KUKA KRL program: MyProgram_146().src

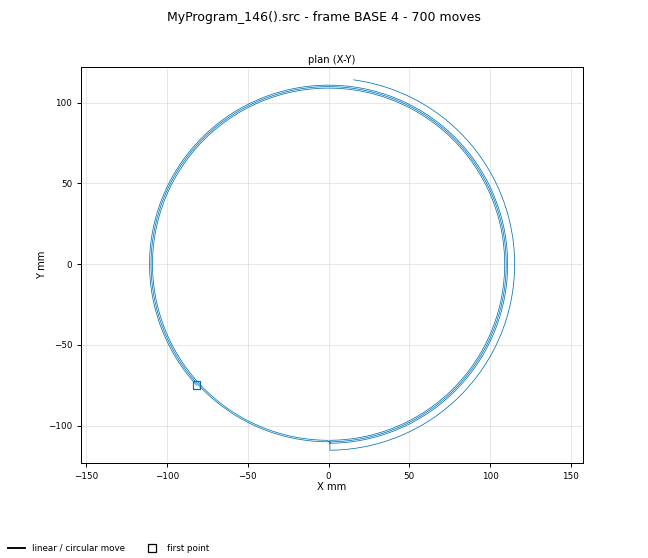
[picture p0: tool path of MyProgram_146().src in frame BASE 4, 700 of 700 moves have a stored position in this frame; points joined in program order, loops and branches not executed]
&ACCESS RVP
&REL 1
&PARAM TEMPLATE = C:\KRC\Roboter\Template\vorgabe
&PARAM EDITMASK = *
DEF MyProgram_146()
; ---- Setting reference (Base) ----
$BASE = BASE_DATA[4]

; --------------------------
; ---- Setting tool (TCP) ----
$TOOL = TOOL_DATA[3]
; --------------------------

$VEL.CP = VEL_APROX_PRINT
Startdeposition()
$VEL.CP = VEL_PRINT
LIN {X -81.7573,Y -74.8316,Z 115,A -141.7153,B 24.9501,C -1.6313,E1 24.8814,E2 227.6019} C_DIS
LIN {X -84.7818,Y -71.3896,Z 115,A -144.2948,B 24.9503,C -1.6285,E1 24.8767,E2 230.1997} C_DIS
LIN {X -86.9243,Y -68.7617,Z 115,A -146.5277,B 24.9512,C -1.6142,E1 24.8727,E2 232.4772} C_DIS
LIN {X -89.3897,Y -65.5248,Z 115,A -148.18,B 24.9498,C -1.6368,E1 24.87,E2 234.0837} C_DIS
LIN {X -91.5986,Y -62.4003,Z 115,A -150.3386,B 24.9499,C -1.6348,E1 24.8666,E2 236.2576} C_DIS
LIN {X -94.0442,Y -58.649,Z 115,A -152.3948,B 24.9489,C -1.6509,E1 24.8635,E2 238.286} C_DIS
LIN {X -96.0088,Y -55.3746,Z 115,A -154.4318,B 24.9488,C -1.6537,E1 24.8607,E2 240.3268} C_DIS
LIN {X -98.582,Y -50.6523,Z 115,A -157.2694,B 24.9484,C -1.6592,E1 24.8569,E2 243.1663} C_DIS
LIN {X -100.3639,Y -47.023,Z 115,A -159.3857,B 24.9481,C -1.6641,E1 24.8544,E2 245.2824} C_DIS
LIN {X -102.0957,Y -43.1333,Z 115,A -161.4118,B 24.9473,C -1.6772,E1 24.8521,E2 247.2885} C_DIS
LIN {X -103.2527,Y -40.2858,Z 115,A -163.0662,B 24.9472,C -1.6793,E1 24.8504,E2 248.9471} C_DIS
LIN {X -104.2802,Y -37.548,Z 115,A -164.6637,B 24.9471,C -1.6805,E1 24.8489,E2 250.5507} C_DIS
LIN {X -105.4561,Y -34.1032,Z 115,A -166.5332,B 24.9467,C -1.6867,E1 24.8472,E2 252.4164} C_DIS
LIN {X -107.1592,Y -28.3073,Z 115,A -169.7153,B 24.9462,C -1.6939,E1 24.8448,E2 255.5995} C_DIS
LIN {X -108.4327,Y -22.9525,Z 115,A -172.6096,B 24.9458,C -1.7009,E1 24.843,E2 258.4941} C_DIS
LIN {X -108.951,Y -20.3482,Z 115,A -173.8603,B 24.9452,C -1.7099,E1 24.8423,E2 259.7309} C_DIS
LIN {X -109.5336,Y -16.923,Z 115,A -175.6733,B 24.9449,C -1.7149,E1 24.8415,E2 261.5426} C_DIS
LIN {X -110.023,Y -13.3864,Z 115,A -177.655,B 24.9449,C -1.7156,E1 24.8408,E2 263.5345} C_DIS
LIN {X -110.406,Y -9.7333,Z 115,A -179.5845,B 24.9445,C -1.7206,E1 24.8403,E2 265.4638} C_DIS
LIN {X -110.6566,Y -6.2558,Z 115,A 178.7094,B 24.9439,C -1.73,E1 24.84,E2 267.1575} C_DIS
LIN {X -110.8019,Y -2.7097,Z 115,A 176.7644,B 24.9438,C -1.7318,E1 24.8398,E2 269.1101} C_DIS
LIN {X -110.8276,Y 1.2801,Z 115,A 174.684,B 24.9434,C -1.7378,E1 24.8398,E2 271.1887} C_DIS
LIN {X -110.7364,Y 4.6333,Z 115,A 173.0527,B 24.9428,C -1.7473,E1 24.84,E2 272.807} C_DIS
LIN {X -110.534,Y 8.1638,Z 115,A 171.0925,B 24.9428,C -1.7483,E1 24.8403,E2 274.7769} C_DIS
LIN {X -110.2005,Y 11.8298,Z 115,A 169.1643,B 24.9424,C -1.7535,E1 24.8409,E2 276.7041} C_DIS
LIN {X -109.6262,Y 16.3247,Z 115,A 166.4672,B 24.9428,C -1.7477,E1 24.8419,E2 279.431} C_DIS
LIN {X -109.0594,Y 19.7502,Z 115,A 164.6359,B 24.9425,C -1.7522,E1 24.8428,E2 281.2625} C_DIS
LIN {X -108.342,Y 23.3687,Z 115,A 163.4659,B 24.9402,C -1.7861,E1 24.8435,E2 282.3586} C_DIS
LIN {X -106.823,Y 29.5519,Z 115,A 159.9331,B 24.9402,C -1.7874,E1 24.8459,E2 285.909} C_DIS
LIN {X -105.5105,Y 33.9351,Z 115,A 157.4846,B 24.9398,C -1.7917,E1 24.8479,E2 288.3612} C_DIS
LIN {X -104.4742,Y 37.0035,Z 115,A 155.7145,B 24.9398,C -1.7934,E1 24.8495,E2 290.1375} C_DIS
LIN {X -103.1875,Y 40.4518,Z 115,A 154.094,B 24.9386,C -1.81,E1 24.8511,E2 291.7276} C_DIS
LIN {X -100.9318,Y 45.7915,Z 115,A 150.7623,B 24.9388,C -1.8064,E1 24.8548,E2 295.0862} C_DIS
LIN {X -99.2356,Y 49.3592,Z 115,A 148.8447,B 24.9381,C -1.8172,E1 24.8571,E2 296.9882} C_DIS
LIN {X -97.7685,Y 52.2085,Z 115,A 147.0374,B 24.9381,C -1.8164,E1 24.8595,E2 298.8072} C_DIS
LIN {X -96.07,Y 55.2682,Z 115,A 145.1429,B 24.9381,C -1.8185,E1 24.8621,E2 300.7066} C_DIS
LIN {X -92.0549,Y 61.7265,Z 115,A 141.3379,B 24.9369,C -1.8344,E1 24.8678,E2 304.4929} C_DIS
LIN {X -90.3878,Y 64.1416,Z 115,A 139.117,B 24.9385,C -1.812,E1 24.8715,E2 306.7782} C_DIS
LIN {X -87.5356,Y 67.9832,Z 115,A 137.571,B 24.9356,C -1.8539,E1 24.8739,E2 308.2317} C_DIS
LIN {X -83.6667,Y 72.6909,Z 115,A 134.1861,B 24.9356,C -1.8531,E1 24.88,E2 311.6341} C_DIS
LIN {X -79.1475,Y 77.5878,Z 115,A 129.9553,B 24.9371,C -1.8317,E1 24.8883,E2 315.9343} C_DIS
LIN {X -75.6083,Y 81.0407,Z 115,A 128.058,B 24.9349,C -1.8629,E1 24.892,E2 317.765} C_DIS
LIN {X -70.4692,Y 85.5472,Z 115,A 123.8886,B 24.9361,C -1.8465,E1 24.901,E2 321.9897} C_DIS
LIN {X -66.7924,Y 88.4469,Z 115,A 122.3719,B 24.9333,C -1.8865,E1 24.9041,E2 323.4166} C_DIS
LIN {X -62.2506,Y 91.7,Z 115,A 119.1568,B 24.9338,C -1.8796,E1 24.9115,E2 326.6592} C_DIS
LIN {X -58.8492,Y 93.9192,Z 115,A 117.1695,B 24.9332,C -1.888,E1 24.9162,E2 328.6329} C_DIS
LIN {X -56.138,Y 95.5648,Z 115,A 115.439,B 24.9332,C -1.8874,E1 24.9203,E2 330.37} C_DIS
LIN {X -53.5767,Y 97.0249,Z 115,A 113.3768,B 24.9345,C -1.8691,E1 24.9255,E2 332.4818} C_DIS
LIN {X -49.7768,Y 99.0286,Z 115,A 111.6694,B 24.9328,C -1.8928,E1 24.9296,E2 334.1375} C_DIS
LIN {X -46.6238,Y 100.5498,Z 115,A 110.0445,B 24.9321,C -1.9029,E1 24.9337,E2 335.7423} C_DIS
LIN {X -40.112,Y 103.321,Z 115,A 106.2146,B 24.9322,C -1.9013,E1 24.9436,E2 339.5847} C_DIS
LIN {X -35.6021,Y 104.9597,Z 115,A 103.1863,B 24.9335,C -1.8828,E1 24.9517,E2 342.6629} C_DIS
LIN {X -31.5857,Y 106.2373,Z 115,A 101.555,B 24.9318,C -1.907,E1 24.9559,E2 344.2396} C_DIS
LIN {X -26.5277,Y 107.6121,Z 115,A 98.9611,B 24.9313,C -1.9143,E1 24.9629,E2 346.82} C_DIS
LIN {X -23.7708,Y 108.2542,Z 115,A 97.4433,B 24.9313,C -1.9135,E1 24.967,E2 348.3417} C_DIS
LIN {X -20.5939,Y 108.9038,Z 115,A 95.6798,B 24.9315,C -1.9113,E1 24.9718,E2 350.1123} C_DIS
LIN {X -16.923,Y 109.5336,Z 115,A 93.8834,B 24.931,C -1.9179,E1 24.9768,E2 351.8948} C_DIS
LIN {X -13.8535,Y 109.9647,Z 115,A 92.371,B 24.9307,C -1.9226,E1 24.9809,E2 353.3972} C_DIS
LIN {X -10.0487,Y 110.3769,Z 115,A 90.2727,B 24.931,C -1.9187,E1 24.9868,E2 355.5058} C_DIS
LIN {X -6.4735,Y 110.6446,Z 115,A 88.3325,B 24.9312,C -1.916,E1 24.9922,E2 357.4533} C_DIS
LIN {X -3.889,Y 110.7661,Z 115,A 86.8091,B 24.9317,C -1.9088,E1 24.9965,E2 358.9939} C_DIS
LIN {X 0.2371,Y 110.8339,Z 115,A 84.7338,B 24.9315,C -1.9116,E1 25.0023,E2 361.0626} C_DIS
LIN {X 4.4661,Y 110.7436,Z 115,A 82.7039,B 24.931,C -1.9183,E1 25.0079,E2 363.0763} C_DIS
LIN {X 7.7943,Y 110.5593,Z 115,A 80.9252,B 24.9312,C -1.916,E1 25.0129,E2 364.8597} C_DIS
LIN {X 11.1548,Y 110.2712,Z 115,A 79.1362,B 24.9313,C -1.9139,E1 25.0178,E2 366.6525} C_DIS
LIN {X 15.2675,Y 109.7771,Z 115,A 77.1238,B 24.931,C -1.9188,E1 25.0234,E2 368.6517} C_DIS
LIN {X 18.2241,Y 109.3247,Z 115,A 75.5914,B 24.931,C -1.9188,E1 25.0276,E2 370.1824} C_DIS
LIN {X 21.6751,Y 108.6949,Z 115,A 73.7246,B 24.9312,C -1.9159,E1 25.0327,E2 372.0541} C_DIS
LIN {X 24.7884,Y 108.0258,Z 115,A 72.0718,B 24.9312,C -1.9148,E1 25.0372,E2 373.7073} C_DIS
LIN {X 28.6398,Y 107.0694,Z 115,A 69.2783,B 24.9336,C -1.8827,E1 25.045,E2 376.5725} C_DIS
LIN {X 33.4912,Y 105.6541,Z 115,A 67.5311,B 24.9311,C -1.9167,E1 25.0494,E2 378.236} C_DIS
LIN {X 37.5394,Y 104.2834,Z 115,A 65.2305,B 24.9315,C -1.9109,E1 25.0555,E2 380.5457} C_DIS
LIN {X 40.4462,Y 103.1897,Z 115,A 63.6357,B 24.9316,C -1.9098,E1 25.0597,E2 382.1396} C_DIS
LIN {X 43.8995,Y 101.7695,Z 115,A 61.6688,B 24.9319,C -1.9062,E1 25.0647,E2 384.1106} C_DIS
LIN {X 46.9047,Y 100.419,Z 115,A 59.6955,B 24.9328,C -1.8927,E1 25.0698,E2 386.1106} C_DIS
LIN {X 51.8783,Y 97.9424,Z 115,A 56.88,B 24.9329,C -1.8914,E1 25.0768,E2 388.9215} C_DIS
LIN {X 56.568,Y 95.3106,Z 115,A 54.359,B 24.9324,C -1.8984,E1 25.0828,E2 391.4183} C_DIS
LIN {X 59.6032,Y 93.4429,Z 115,A 52.5572,B 24.9325,C -1.8973,E1 25.0871,E2 393.2171} C_DIS
LIN {X 62.4108,Y 91.5915,Z 115,A 50.819,B 24.9327,C -1.8944,E1 25.0911,E2 394.9561} C_DIS
LIN {X 65.368,Y 89.5045,Z 115,A 49.1942,B 24.9322,C -1.9018,E1 25.0948,E2 396.5578} C_DIS
LIN {X 67.3354,Y 88.0347,Z 115,A 47.6455,B 24.9332,C -1.8875,E1 25.0983,E2 398.1348} C_DIS
LIN {X 69.5282,Y 86.313,Z 115,A 46.1298,B 24.9336,C -1.8816,E1 25.1016,E2 399.6588} C_DIS
LIN {X 72.7487,Y 83.6163,Z 115,A 44.0933,B 24.9336,C -1.8832,E1 25.1059,E2 401.6836} C_DIS
LIN {X 76.092,Y 80.5858,Z 115,A 41.7552,B 24.9339,C -1.8782,E1 25.1107,E2 404.024} C_DIS
LIN {X 78.6426,Y 78.0989,Z 115,A 40.1113,B 24.9335,C -1.8829,E1 25.114,E2 405.65} C_DIS
LIN {X 82.0766,Y 74.4837,Z 115,A 37.2578,B 24.9348,C -1.865,E1 25.1195,E2 408.5332} C_DIS
LIN {X 84.4274,Y 71.8056,Z 115,A 35.5078,B 24.9348,C -1.8648,E1 25.1226,E2 410.2757} C_DIS
LIN {X 86.8535,Y 68.8514,Z 115,A 33.7446,B 24.9345,C -1.8694,E1 25.1257,E2 412.0199} C_DIS
LIN {X 89.0528,Y 65.9849,Z 115,A 31.6509,B 24.9355,C -1.8548,E1 25.1293,E2 414.138} C_DIS
LIN {X 90.925,Y 63.3772,Z 115,A 30.0629,B 24.9355,C -1.8538,E1 25.1318,E2 415.7207} C_DIS
LIN {X 92.9023,Y 60.4452,Z 115,A 28.1746,B 24.9361,C -1.8464,E1 25.1348,E2 417.6171} C_DIS
LIN {X 95.8988,Y 55.566,Z 115,A 24.8642,B 24.9377,C -1.8231,E1 25.1396,E2 420.9656} C_DIS
LIN {X 97.6104,Y 52.5013,Z 115,A 23.4849,B 24.9367,C -1.8373,E1 25.1414,E2 422.3042} C_DIS
LIN {X 99.1431,Y 49.5458,Z 115,A 21.7653,B 24.9371,C -1.8325,E1 25.1435,E2 424.0259} C_DIS
LIN {X 100.5688,Y 46.5828,Z 115,A 20.112,B 24.9372,C -1.8297,E1 25.1455,E2 425.6768} C_DIS
LIN {X 102.0077,Y 43.3421,Z 115,A 18.1675,B 24.9379,C -1.8195,E1 25.1477,E2 427.6349} C_DIS
LIN {X 104.8831,Y 35.8293,Z 115,A 14.3206,B 24.9379,C -1.821,E1 25.1514,E2 431.4568} C_DIS
LIN {X 106.5349,Y 30.5691,Z 115,A 11.3263,B 24.9389,C -1.8058,E1 25.1539,E2 434.4698} C_DIS
LIN {X 107.3131,Y 27.7113,Z 115,A 9.7848,B 24.9392,C -1.8007,E1 25.155,E2 436.0146} C_DIS
LIN {X 108.1774,Y 24.1233,Z 115,A 7.8397,B 24.9397,C -1.793,E1 25.1562,E2 437.9664} C_DIS
LIN {X 108.884,Y 20.697,Z 115,A 5.995,B 24.9402,C -1.7857,E1 25.1572,E2 439.8175} C_DIS
LIN {X 109.5415,Y 16.8721,Z 115,A 4.1105,B 24.9402,C -1.7848,E1 25.1581,E2 441.6932} C_DIS
LIN {X 110.0434,Y 13.2119,Z 115,A 2.0838,B 24.9411,C -1.7735,E1 25.1588,E2 443.7346} C_DIS
LIN {X 110.4516,Y 9.1978,Z 115,A 0.0951,B 24.9412,C -1.7711,E1 25.1593,E2 445.7171} C_DIS
LIN {X 110.6876,Y 5.6966,Z 115,A -1.8682,B 24.942,C -1.7586,E1 25.1597,E2 447.6983} C_DIS
LIN {X 110.8179,Y 1.8536,Z 115,A -3.8981,B 24.9426,C -1.7502,E1 25.1597,E2 449.7357} C_DIS
LIN {X 110.7895,Y -3.1254,Z 115,A -6.2103,B 24.9424,C -1.7536,E1 25.1597,E2 452.0262} C_DIS
LIN {X 110.6672,Y -6.0644,Z 115,A -8.3066,B 24.9444,C -1.7229,E1 25.1594,E2 454.1824} C_DIS
LIN {X 110.3562,Y -10.2724,Z 115,A -9.8676,B 24.943,C -1.7435,E1 25.159,E2 455.6856} C_DIS
LIN {X 109.9421,Y -14.0283,Z 115,A -11.804,B 24.9434,C -1.7379,E1 25.1584,E2 457.6237} C_DIS
LIN {X 109.5152,Y -17.0426,Z 115,A -13.3694,B 24.9437,C -1.7332,E1 25.1577,E2 459.1911} C_DIS
LIN {X 108.8663,Y -20.7887,Z 115,A -15.2807,B 24.944,C -1.7293,E1 25.1568,E2 461.1005} C_DIS
LIN {X 108.2063,Y -23.9905,Z 115,A -17.0194,B 24.9445,C -1.7216,E1 25.1558,E2 462.8471} C_DIS
LIN {X 107.4311,Y -27.2525,Z 115,A -18.7555,B 24.9448,C -1.7159,E1 25.1546,E2 464.5865} C_DIS
LIN {X 106.7672,Y -29.7492,Z 115,A -20.4664,B 24.9462,C -1.6949,E1 25.1533,E2 466.3373} C_DIS
LIN {X 105.817,Y -32.9666,Z 115,A -21.8898,B 24.9456,C -1.7033,E1 25.1521,E2 467.7328} C_DIS
LIN {X 104.6176,Y -36.5948,Z 115,A -23.6513,B 24.9454,C -1.7067,E1 25.1506,E2 469.4764} C_DIS
LIN {X 103.7534,Y -38.9785,Z 115,A -25.1912,B 24.9463,C -1.6923,E1 25.1491,E2 471.0416} C_DIS
LIN {X 102.2201,Y -42.8382,Z 115,A -27.182,B 24.9463,C -1.6926,E1 25.147,E2 473.0206} C_DIS
LIN {X 100.7679,Y -46.1551,Z 115,A -28.9646,B 24.9464,C -1.6909,E1 25.1449,E2 474.7976} C_DIS
LIN {X 98.7191,Y -50.3841,Z 115,A -31.9765,B 24.9485,C -1.6576,E1 25.1411,E2 477.8719} C_DIS
LIN {X 96.8713,Y -53.8517,Z 115,A -33.4559,B 24.9474,C -1.6762,E1 25.1392,E2 479.2998} C_DIS
LIN {X 95.5696,Y -56.1298,Z 115,A -35.2243,B 24.9487,C -1.6538,E1 25.1367,E2 481.1118} C_DIS
LIN {X 93.7863,Y -59.0619,Z 115,A -36.7745,B 24.9484,C -1.6587,E1 25.1344,E2 482.6427} C_DIS
LIN {X 90.7878,Y -63.5747,Z 115,A -39.4423,B 24.9486,C -1.6567,E1 25.1302,E2 485.3019} C_DIS
LIN {X 88.6944,Y -66.463,Z 115,A -41.1973,B 24.9486,C -1.6556,E1 25.1273,E2 487.0511} C_DIS
LIN {X 86.5166,Y -69.2771,Z 115,A -43.1288,B 24.9492,C -1.6465,E1 25.1239,E2 488.995} C_DIS
LIN {X 84.2505,Y -72.0131,Z 115,A -44.9007,B 24.9493,C -1.6446,E1 25.1208,E2 490.7634} C_DIS
LIN {X 81.7575,Y -74.8315,Z 115,A -46.8119,B 24.9495,C -1.6411,E1 25.1172,E2 492.6742} C_DIS
LIN {X 79.0371,Y -77.6995,Z 115,A -48.8035,B 24.9497,C -1.6383,E1 25.1133,E2 494.6639} C_DIS
LIN {X 76.7863,Y -79.9244,Z 115,A -50.4986,B 24.9501,C -1.6317,E1 25.1099,E2 496.3675} C_DIS
LIN {X 74.0477,Y -82.468,Z 115,A -52.3792,B 24.9502,C -1.6294,E1 25.1061,E2 498.2458} C_DIS
LIN {X 71.2837,Y -84.8704,Z 115,A -54.3202,B 24.9506,C -1.623,E1 25.1019,E2 500.1946} C_DIS
LIN {X 68.6576,Y -87.0066,Z 115,A -55.9786,B 24.9506,C -1.6231,E1 25.0983,E2 501.8463} C_DIS
LIN {X 65.6879,Y -89.2702,Z 115,A -57.9458,B 24.951,C -1.6174,E1 25.0939,E2 503.82} C_DIS
LIN {X 62.8535,Y -91.2891,Z 115,A -59.5768,B 24.9508,C -1.6211,E1 25.0902,E2 505.4367} C_DIS
LIN {X 60.4943,Y -92.87,Z 115,A -62.3586,B 24.9543,C -1.5612,E1 25.0834,E2 508.3508} C_DIS
LIN {X 54.7496,Y -96.368,Z 115,A -65.2533,B 24.9532,C -1.5799,E1 25.0765,E2 511.1928} C_DIS
LIN {X 50.9504,Y -98.4297,Z 115,A -66.9022,B 24.952,C -1.6013,E1 25.0726,E2 512.7863} C_DIS
LIN {X 47.5157,Y -100.1327,Z 115,A -68.9366,B 24.9523,C -1.5958,E1 25.0674,E2 514.8283} C_DIS
LIN {X 44.9116,Y -101.3283,Z 115,A -70.6659,B 24.9531,C -1.5828,E1 25.063,E2 516.584} C_DIS
LIN {X 40.4823,Y -103.1756,Z 115,A -72.88,B 24.9526,C -1.5908,E1 25.0573,E2 518.7742} C_DIS
LIN {X 35.6279,Y -104.951,Z 115,A -75.4422,B 24.9526,C -1.592,E1 25.0506,E2 521.3284} C_DIS
LIN {X 32.2394,Y -106.0419,Z 115,A -77.3857,B 24.9529,C -1.5854,E1 25.0454,E2 523.2841} C_DIS
LIN {X 28.9748,Y -106.9789,Z 115,A -79.0339,B 24.9527,C -1.5881,E1 25.041,E2 524.9231} C_DIS
LIN {X 25.2858,Y -107.9109,Z 115,A -81.0187,B 24.9529,C -1.5854,E1 25.0356,E2 526.9115} C_DIS
LIN {X 22.1944,Y -108.5883,Z 115,A -82.4818,B 24.9526,C -1.5913,E1 25.0316,E2 528.3588} C_DIS
LIN {X 18.4966,Y -109.2791,Z 115,A -84.5679,B 24.953,C -1.5837,E1 25.0258,E2 530.4605} C_DIS
LIN {X 15.2443,Y -109.7804,Z 115,A -86.3172,B 24.9532,C -1.5804,E1 25.021,E2 532.2159} C_DIS
LIN {X 12.7171,Y -110.1014,Z 115,A -87.747,B 24.9535,C -1.5749,E1 25.017,E2 533.6579} C_DIS
LIN {X 6.9538,Y -110.6161,Z 115,A -90.5923,B 24.9533,C -1.5795,E1 25.0091,E2 536.4906} C_DIS
LIN {X 3.5153,Y -110.7775,Z 115,A -92.3395,B 24.9533,C -1.5803,E1 25.0042,E2 538.2356} C_DIS
LIN {X 0.7828,Y -110.8248,Z 115,A -93.8199,B 24.9533,C -1.5771,E1 25.0001,E2 539.7233} C_DIS
Enddeposition()
LIN {X 0.7828,Y -110.8248,Z 115,A -93.8199,B 24.9533,C -1.5771,E1 25.0001,E2 539.7233} C_DIS
Startdeposition()
$VEL.CP = VEL_PRINT
LIN {X 1.4576,Y -109.912,Z 115,A -92.785,B 24.9507,C -1.6218,E1 25.0033,E2 538.5826} C_DIS
LIN {X 4.6673,Y -109.8211,Z 115,A -91.0978,B 24.9507,C -1.623,E1 25.008,E2 536.893} C_DIS
LIN {X 7.5586,Y -109.6601,Z 115,A -89.4834,B 24.9503,C -1.6281,E1 25.0125,E2 535.2672} C_DIS
LIN {X 11.1892,Y -109.3495,Z 115,A -87.5115,B 24.9501,C -1.6322,E1 25.018,E2 533.2868} C_DIS
LIN {X 14.8057,Y -108.9205,Z 115,A -85.5197,B 24.9498,C -1.6373,E1 25.0236,E2 531.2843} C_DIS
LIN {X 18.9126,Y -108.2823,Z 115,A -83.6444,B 24.9504,C -1.6265,E1 25.0287,E2 529.4365} C_DIS
LIN {X 22.0138,Y -107.6933,Z 115,A -81.8972,B 24.9501,C -1.6323,E1 25.0335,E2 527.6777} C_DIS
LIN {X 25.453,Y -106.9345,Z 115,A -79.9474,B 24.9497,C -1.6389,E1 25.0388,E2 525.7149} C_DIS
LIN {X 29.0229,Y -106.0201,Z 115,A -78.0363,B 24.9496,C -1.6406,E1 25.044,E2 523.8029} C_DIS
LIN {X 31.771,Y -105.2299,Z 115,A -76.3612,B 24.949,C -1.6503,E1 25.0485,E2 522.1078} C_DIS
LIN {X 36.3044,Y -103.7519,Z 115,A -73.5988,B 24.948,C -1.6655,E1 25.0559,E2 519.3147} C_DIS
LIN {X 40.1137,Y -102.3394,Z 115,A -71.6969,B 24.9484,C -1.659,E1 25.0608,E2 517.4325} C_DIS
LIN {X 43.1125,Y -101.1137,Z 115,A -70.4315,B 24.9494,C -1.6431,E1 25.0639,E2 516.2078} C_DIS
LIN {X 45.8081,Y -99.9224,Z 115,A -68.7252,B 24.9488,C -1.6528,E1 25.0683,E2 514.4827} C_DIS
LIN {X 48.7959,Y -98.4957,Z 115,A -67.0984,B 24.9488,C -1.6514,E1 25.0724,E2 512.8636} C_DIS
LIN {X 51.1648,Y -97.2863,Z 115,A -65.5915,B 24.9484,C -1.659,E1 25.0761,E2 511.3429} C_DIS
LIN {X 54.8199,Y -95.2745,Z 115,A -63.5622,B 24.9486,C -1.6565,E1 25.0811,E2 509.3255} C_DIS
LIN {X 58.1891,Y -93.255,Z 115,A -61.7581,B 24.949,C -1.6497,E1 25.0853,E2 507.5431} C_DIS
LIN {X 62.6693,Y -90.3051,Z 115,A -58.7684,B 24.9481,C -1.6637,E1 25.0923,E2 504.5302} C_DIS
LIN {X 65.4015,Y -88.3483,Z 115,A -56.9115,B 24.9476,C -1.672,E1 25.0965,E2 502.6603} C_DIS
LIN {X 68.1462,Y -86.247,Z 115,A -55.2231,B 24.9476,C -1.671,E1 25.1002,E2 500.9807} C_DIS
LIN {X 71.0085,Y -83.9069,Z 115,A -53.25,B 24.9473,C -1.6773,E1 25.1045,E2 499.0001} C_DIS
LIN {X 73.7158,Y -81.5397,Z 115,A -51.3437,B 24.9469,C -1.6831,E1 25.1085,E2 497.0877} C_DIS
LIN {X 76.198,Y -79.2233,Z 115,A -49.6701,B 24.9469,C -1.6831,E1 25.1118,E2 495.421} C_DIS
LIN {X 78.6653,Y -76.7767,Z 115,A -47.7296,B 24.9463,C -1.6933,E1 25.1157,E2 493.4647} C_DIS
LIN {X 81.2752,Y -74.0066,Z 115,A -45.7835,B 24.9461,C -1.6967,E1 25.1194,E2 491.5192} C_DIS
LIN {X 83.5964,Y -71.3731,Z 115,A -44.0758,B 24.9461,C -1.696,E1 25.1225,E2 489.8208} C_DIS
LIN {X 85.812,Y -68.6964,Z 115,A -42.1422,B 24.9454,C -1.7063,E1 25.1259,E2 487.8719} C_DIS
LIN {X 88.352,Y -65.3964,Z 115,A -40.0792,B 24.9454,C -1.7074,E1 25.1294,E2 485.8161} C_DIS
LIN {X 90.1847,Y -62.8426,Z 115,A -37.7884,B 24.9432,C -1.7414,E1 25.1331,E2 483.4563} C_DIS
LIN {X 92.7748,Y -58.9537,Z 115,A -36.0541,B 24.9448,C -1.7167,E1 25.1357,E2 481.7891} C_DIS
LIN {X 94.7217,Y -55.77,Z 115,A -34.1518,B 24.9445,C -1.7204,E1 25.1384,E2 479.8878} C_DIS
LIN {X 96.4518,Y -52.7223,Z 115,A -32.2608,B 24.944,C -1.7287,E1 25.141,E2 477.9871} C_DIS
LIN {X 97.7068,Y -50.3585,Z 115,A -30.3408,B 24.9422,C -1.7566,E1 25.1435,E2 476.0115} C_DIS
LIN {X 99.537,Y -46.6359,Z 115,A -28.7858,B 24.9435,C -1.7356,E1 25.1453,E2 474.5142} C_DIS
LIN {X 100.9223,Y -43.558,Z 115,A -27.0904,B 24.9434,C -1.7381,E1 25.1472,E2 472.8222} C_DIS
LIN {X 102.2903,Y -40.2388,Z 115,A -25.4454,B 24.9437,C -1.7338,E1 25.1489,E2 471.1965} C_DIS
LIN {X 103.8515,Y -36.0204,Z 115,A -22.9448,B 24.9427,C -1.7481,E1 25.1513,E2 468.6762} C_DIS
LIN {X 105.806,Y -29.7921,Z 115,A -19.4702,B 24.9418,C -1.7621,E1 25.1542,E2 465.1884} C_DIS
LIN {X 106.6681,Y -26.5449,Z 115,A -17.653,B 24.9412,C -1.7706,E1 25.1554,E2 463.3615} C_DIS
LIN {X 107.4491,Y -23.1778,Z 115,A -15.8685,B 24.9409,C -1.7757,E1 25.1565,E2 461.5754} C_DIS
LIN {X 108.1717,Y -19.5282,Z 115,A -14.0375,B 24.9409,C -1.777,E1 25.1575,E2 459.7519} C_DIS
LIN {X 108.6569,Y -16.6183,Z 115,A -12.448,B 24.9403,C -1.7844,E1 25.1582,E2 458.1545} C_DIS
LIN {X 109.1437,Y -13.0455,Z 115,A -10.6244,B 24.9401,C -1.788,E1 25.1588,E2 456.3332} C_DIS
LIN {X 109.4667,Y -9.975,Z 115,A -9.2078,B 24.9403,C -1.7845,E1 25.1592,E2 454.9332} C_DIS
LIN {X 109.6979,Y -6.9997,Z 115,A -7.3761,B 24.9391,C -1.802,E1 25.1596,E2 453.071} C_DIS
LIN {X 109.859,Y -3.6799,Z 115,A -5.9668,B 24.9397,C -1.7931,E1 25.1597,E2 451.6912} C_DIS
LIN {X 109.9189,Y -0.535,Z 115,A -4.0353,B 24.9385,C -1.8116,E1 25.1597,E2 449.7276} C_DIS
LIN {X 109.8898,Y 2.662,Z 115,A -2.2548,B 24.9378,C -1.8221,E1 25.1597,E2 447.9327} C_DIS
LIN {X 109.693,Y 7.0722,Z 115,A -0.2487,B 24.9382,C -1.8162,E1 25.1594,E2 445.9525} C_DIS
LIN {X 109.43,Y 10.3734,Z 115,A 1.6087,B 24.9374,C -1.8277,E1 25.1589,E2 444.079} C_DIS
LIN {X 109.0112,Y 14.1072,Z 115,A 3.4891,B 24.9372,C -1.8305,E1 25.1583,E2 442.2033} C_DIS
LIN {X 108.4782,Y 17.7505,Z 115,A 5.2562,B 24.9372,C -1.8297,E1 25.1576,E2 440.4483} C_DIS
LIN {X 108.0255,Y 20.3262,Z 115,A 6.7767,B 24.9365,C -1.8411,E1 25.1568,E2 438.9099} C_DIS
LIN {X 107.3718,Y 23.532,Z 115,A 8.436,B 24.9362,C -1.8444,E1 25.1558,E2 437.2525} C_DIS
LIN {X 106.5272,Y 27.1013,Z 115,A 10.2668,B 24.9361,C -1.8467,E1 25.1546,E2 435.4269} C_DIS
LIN {X 105.6647,Y 30.2908,Z 115,A 12.2896,B 24.9348,C -1.8655,E1 25.1531,E2 433.3714} C_DIS
LIN {X 104.2206,Y 34.9364,Z 115,A 14.5101,B 24.9352,C -1.859,E1 25.1512,E2 431.1787} C_DIS
LIN {X 103.121,Y 38.0617,Z 115,A 16.0603,B 24.9354,C -1.8562,E1 25.1497,E2 429.6437} C_DIS
LIN {X 101.7737,Y 41.528,Z 115,A 18.2079,B 24.9344,C -1.8713,E1 25.1475,E2 427.4725} C_DIS
LIN {X 100.48,Y 44.5717,Z 115,A 19.8573,B 24.9342,C -1.8729,E1 25.1457,E2 425.8282} C_DIS
LIN {X 99.0826,Y 47.5931,Z 115,A 21.6292,B 24.9338,C -1.8795,E1 25.1436,E2 424.0504} C_DIS
LIN {X 97.4102,Y 50.9296,Z 115,A 23.5402,B 24.9335,C -1.8834,E1 25.1411,E2 422.1403} C_DIS
LIN {X 95.6169,Y 54.2241,Z 115,A 25.6008,B 24.9328,C -1.8934,E1 25.1383,E2 420.0668} C_DIS
LIN {X 93.0934,Y 58.4477,Z 115,A 28.1085,B 24.9325,C -1.8978,E1 25.1347,E2 417.5616} C_DIS
LIN {X 90.9639,Y 61.7093,Z 115,A 30.0964,B 24.9322,C -1.9011,E1 25.1316,E2 415.5756} C_DIS
LIN {X 88.7346,Y 64.8739,Z 115,A 32.009,B 24.9322,C -1.9016,E1 25.1285,E2 413.6713} C_DIS
LIN {X 86.9899,Y 67.1954,Z 115,A 33.6534,B 24.9315,C -1.9111,E1 25.1257,E2 412.0123} C_DIS
LIN {X 84.5713,Y 70.215,Z 115,A 35.5552,B 24.9315,C -1.9108,E1 25.1224,E2 410.1199} C_DIS
LIN {X 82.4432,Y 72.7038,Z 115,A 37.3732,B 24.9309,C -1.9196,E1 25.119,E2 408.2893} C_DIS
LIN {X 79.5768,Y 75.8311,Z 115,A 39.5874,B 24.9306,C -1.9247,E1 25.1148,E2 406.0728} C_DIS
LIN {X 77.2542,Y 78.1936,Z 115,A 41.2499,B 24.9305,C -1.9256,E1 25.1115,E2 404.4152} C_DIS
LIN {X 74.4224,Y 80.8936,Z 115,A 43.3554,B 24.93,C -1.9327,E1 25.1072,E2 402.3015} C_DIS
LIN {X 71.3363,Y 83.6277,Z 115,A 45.3923,B 24.93,C -1.9321,E1 25.1029,E2 400.2741} C_DIS
LIN {X 68.4491,Y 86.0076,Z 115,A 47.3184,B 24.9298,C -1.9347,E1 25.0988,E2 398.3491} C_DIS
LIN {X 65.461,Y 88.3047,Z 115,A 49.3046,B 24.9295,C -1.9392,E1 25.0943,E2 396.3596} C_DIS
LIN {X 62.7418,Y 90.2547,Z 115,A 51.0231,B 24.9294,C -1.9411,E1 25.0904,E2 394.6426} C_DIS
LIN {X 59.6622,Y 92.32,Z 115,A 52.8973,B 24.9294,C -1.9417,E1 25.0861,E2 392.7732} C_DIS
LIN {X 57.0639,Y 93.9477,Z 115,A 54.595,B 24.9288,C -1.9484,E1 25.082,E2 391.0649} C_DIS
LIN {X 54.0271,Y 95.7276,Z 115,A 56.3632,B 24.9288,C -1.9482,E1 25.0777,E2 389.3025} C_DIS
LIN {X 50.5368,Y 97.6157,Z 115,A 58.5313,B 24.9283,C -1.9552,E1 25.0724,E2 387.1239} C_DIS
LIN {X 46.8685,Y 99.4288,Z 115,A 60.669,B 24.9281,C -1.958,E1 25.067,E2 384.9851} C_DIS
LIN {X 43.3229,Y 101.0248,Z 115,A 62.6639,B 24.9281,C -1.9589,E1 25.0619,E2 382.993} C_DIS
LIN {X 39.9929,Y 102.3868,Z 115,A 64.4856,B 24.9281,C -1.9586,E1 25.0572,E2 381.1761} C_DIS
LIN {X 36.5061,Y 103.6811,Z 115,A 66.5512,B 24.9275,C -1.9658,E1 25.0517,E2 379.0978} C_DIS
LIN {X 32.6587,Y 104.9565,Z 115,A 68.4547,B 24.9281,C -1.9586,E1 25.0467,E2 377.2148} C_DIS
LIN {X 27.8183,Y 106.3429,Z 115,A 71.0376,B 24.9281,C -1.9586,E1 25.0398,E2 374.6361} C_DIS
LIN {X 24.7615,Y 107.0949,Z 115,A 72.8073,B 24.9276,C -1.965,E1 25.0349,E2 372.8539} C_DIS
LIN {X 20.9423,Y 107.9069,Z 115,A 74.8101,B 24.9276,C -1.9645,E1 25.0295,E2 370.8546} C_DIS
LIN {X 17.223,Y 108.5634,Z 115,A 76.8057,B 24.9276,C -1.9663,E1 25.024,E2 368.8568} C_DIS
LIN {X 13.4769,Y 109.0929,Z 115,A 78.8737,B 24.9272,C -1.9707,E1 25.0182,E2 366.78} C_DIS
LIN {X 9.9078,Y 109.4729,Z 115,A 80.5995,B 24.9276,C -1.965,E1 25.0134,E2 365.069} C_DIS
LIN {X 6.572,Y 109.7247,Z 115,A 82.4248,B 24.9274,C -1.9684,E1 25.0083,E2 363.2364} C_DIS
LIN {X 3.0112,Y 109.8795,Z 115,A 84.2279,B 24.9275,C -1.966,E1 25.0033,E2 361.4395} C_DIS
LIN {X -0.6971,Y 109.918,Z 115,A 86.0705,B 24.9278,C -1.9619,E1 24.9982,E2 359.6067} C_DIS
LIN {X -4.0888,Y 109.846,Z 115,A 87.9378,B 24.9276,C -1.9654,E1 24.993,E2 357.7308} C_DIS
LIN {X -6.7639,Y 109.7138,Z 115,A 89.4112,B 24.9274,C -1.968,E1 24.9888,E2 356.2507} C_DIS
LIN {X -9.9457,Y 109.4694,Z 115,A 90.9552,B 24.9278,C -1.9624,E1 24.9846,E2 354.7193} C_DIS
LIN {X -13.7641,Y 109.0556,Z 115,A 92.9952,B 24.9278,C -1.9628,E1 24.9789,E2 352.677} C_DIS
LIN {X -17.0096,Y 108.5964,Z 115,A 94.6382,B 24.928,C -1.959,E1 24.9744,E2 351.0417} C_DIS
LIN {X -20.5547,Y 107.9815,Z 115,A 96.6117,B 24.9279,C -1.9615,E1 24.969,E2 349.0602} C_DIS
LIN {X -24.2773,Y 107.2067,Z 115,A 98.6317,B 24.9279,C -1.9613,E1 24.9634,E2 347.0381} C_DIS
LIN {X -31.4112,Y 105.3367,Z 115,A 102.2476,B 24.9288,C -1.9481,E1 24.9538,E2 343.448} C_DIS
LIN {X -37.5026,Y 103.3249,Z 115,A 105.7374,B 24.9288,C -1.9498,E1 24.9445,E2 339.9477} C_DIS
LIN {X -40.4956,Y 102.1894,Z 115,A 107.3842,B 24.929,C -1.9467,E1 24.9402,E2 338.3049} C_DIS
LIN {X -42.8008,Y 101.2451,Z 115,A 109.0773,B 24.9279,C -1.9605,E1 24.9358,E2 336.5749} C_DIS
LIN {X -45.7367,Y 99.955,Z 115,A 110.548,B 24.9287,C -1.9499,E1 24.9321,E2 335.1257} C_DIS
LIN {X -49.0478,Y 98.3709,Z 115,A 112.2041,B 24.9297,C -1.9367,E1 24.928,E2 333.4968} C_DIS
LIN {X -52.1514,Y 96.7614,Z 115,A 113.9321,B 24.9302,C -1.93,E1 24.9238,E2 331.7801} C_DIS
LIN {X -54.8378,Y 95.2642,Z 115,A 115.7724,B 24.9297,C -1.9365,E1 24.9192,E2 329.919} C_DIS
LIN {X -58.1908,Y 93.2539,Z 115,A 117.884,B 24.9297,C -1.9356,E1 24.9142,E2 327.8029} C_DIS
LIN {X -61.5927,Y 91.0428,Z 115,A 119.7929,B 24.9306,C -1.9234,E1 24.9098,E2 325.9168} C_DIS
LIN {X -64.649,Y 88.8993,Z 115,A 121.8972,B 24.9305,C -1.9256,E1 24.905,E2 323.8} C_DIS
LIN {X -67.2311,Y 86.9624,Z 115,A 123.5771,B 24.9308,C -1.9219,E1 24.9012,E2 322.1227} C_DIS
LIN {X -69.838,Y 84.8846,Z 115,A 125.3774,B 24.9308,C -1.9205,E1 24.8973,E2 320.319} C_DIS
LIN {X -74.5917,Y 80.7383,Z 115,A 128.0676,B 24.933,C -1.8898,E1 24.8919,E2 317.6912} C_DIS
LIN {X -78.7327,Y 76.707,Z 115,A 131.5535,B 24.9323,C -1.9007,E1 24.8848,E2 314.1649} C_DIS
LIN {X -82.7396,Y 72.3645,Z 115,A 134.7436,B 24.9325,C -1.8971,E1 24.8788,E2 310.9691} C_DIS
LIN {X -86.148,Y 68.2714,Z 115,A 137.7478,B 24.9325,C -1.8986,E1 24.8734,E2 307.9475} C_DIS
LIN {X -89.4955,Y 63.8201,Z 115,A 140.4734,B 24.9335,C -1.8838,E1 24.869,E2 305.244} C_DIS
LIN {X -91.3421,Y 61.1507,Z 115,A 142.1937,B 24.9337,C -1.8802,E1 24.8663,E2 303.5238} C_DIS
LIN {X -93.0704,Y 58.4846,Z 115,A 144.1029,B 24.9334,C -1.8852,E1 24.8634,E2 301.593} C_DIS
LIN {X -95.5399,Y 54.3581,Z 115,A 146.2974,B 24.9347,C -1.8659,E1 24.8603,E2 299.4331} C_DIS
LIN {X -96.8757,Y 51.9407,Z 115,A 147.9097,B 24.9346,C -1.8683,E1 24.8582,E2 297.8065} C_DIS
LIN {X -98.2627,Y 49.2661,Z 115,A 149.448,B 24.935,C -1.8624,E1 24.8562,E2 296.2742} C_DIS
LIN {X -99.7209,Y 46.2409,Z 115,A 150.9982,B 24.9359,C -1.8495,E1 24.8544,E2 294.7463} C_DIS
LIN {X -101.0885,Y 43.1722,Z 115,A 153.0295,B 24.9355,C -1.8548,E1 24.8521,E2 292.6911} C_DIS
LIN {X -102.5945,Y 39.4605,Z 115,A 155.1045,B 24.936,C -1.8478,E1 24.85,E2 290.621} C_DIS
LIN {X -103.9354,Y 35.7813,Z 115,A 157.0064,B 24.9368,C -1.8361,E1 24.8482,E2 288.7362} C_DIS
LIN {X -104.9134,Y 32.7979,Z 115,A 158.8392,B 24.9366,C -1.8385,E1 24.8466,E2 286.8874} C_DIS
LIN {X -106.1914,Y 28.3886,Z 115,A 161.4531,B 24.9366,C -1.8393,E1 24.8447,E2 284.2563} C_DIS
LIN {X -107.3459,Y 23.651,Z 115,A 163.7182,B 24.9379,C -1.8206,E1 24.8433,E2 282.0225} C_DIS
LIN {X -108.1049,Y 19.8992,Z 115,A 165.5257,B 24.9388,C -1.8071,E1 24.8423,E2 280.2366} C_DIS
LIN {X -108.8436,Y 15.347,Z 115,A 168.1347,B 24.9388,C -1.8071,E1 24.8412,E2 277.6122} C_DIS
LIN {X -109.2967,Y 11.6936,Z 115,A 170.0634,B 24.9392,C -1.8012,E1 24.8406,E2 275.6859} C_DIS
LIN {X -109.5846,Y 8.5848,Z 115,A 171.7701,B 24.9393,C -1.7989,E1 24.8402,E2 273.9743} C_DIS
LIN {X -109.8073,Y 4.9889,Z 115,A 173.5301,B 24.9401,C -1.7883,E1 24.8399,E2 272.229} C_DIS
LIN {X -109.893,Y 2.4878,Z 115,A 175.0138,B 24.9399,C -1.7909,E1 24.8398,E2 270.7302} C_DIS
LIN {X -109.9129,Y -1.4076,Z 115,A 177.0533,B 24.9403,C -1.7847,E1 24.8398,E2 268.6933} C_DIS
LIN {X -109.82,Y -4.6923,Z 115,A 178.529,B 24.9413,C -1.7701,E1 24.84,E2 267.2434} C_DIS
LIN {X -109.7037,Y -6.9139,Z 115,A 179.9023,B 24.941,C -1.7745,E1 24.8402,E2 265.8514} C_DIS
LIN {X -109.4393,Y -10.2729,Z 115,A -178.3504,B 24.9414,C -1.7685,E1 24.8406,E2 264.1078} C_DIS
LIN {X -108.999,Y -14.201,Z 115,A -176.301,B 24.9418,C -1.7615,E1 24.8413,E2 262.0629} C_DIS
LIN {X -108.5197,Y -17.502,Z 115,A -174.1438,B 24.9411,C -1.7721,E1 24.8423,E2 259.8678} C_DIS
LIN {X -107.9445,Y -20.7468,Z 115,A -172.8703,B 24.9426,C -1.7496,E1 24.8429,E2 258.6402} C_DIS
LIN {X -107.368,Y -23.5493,Z 115,A -170.6741,B 24.9411,C -1.7721,E1 24.8443,E2 256.3775} C_DIS
LIN {X -106.3195,Y -27.9093,Z 115,A -168.9189,B 24.9431,C -1.7424,E1 24.8454,E2 254.683} C_DIS
LIN {X -105.2892,Y -31.5713,Z 115,A -167.0082,B 24.9437,C -1.7336,E1 24.8469,E2 252.7822} C_DIS
LIN {X -104.3697,Y -34.4943,Z 115,A -165.2744,B 24.9437,C -1.734,E1 24.8484,E2 251.0375} C_DIS
LIN {X -103.0344,Y -38.299,Z 115,A -163.1733,B 24.9441,C -1.7277,E1 24.8504,E2 248.9395} C_DIS
LIN {X -101.9108,Y -41.1912,Z 115,A -161.8023,B 24.945,C -1.7135,E1 24.8518,E2 247.5946} C_DIS
LIN {X -100.9472,Y -43.5008,Z 115,A -160.1808,B 24.9444,C -1.7219,E1 24.8536,E2 245.9441} C_DIS
LIN {X -99.043,Y -47.6754,Z 115,A -157.9825,B 24.9454,C -1.7076,E1 24.8562,E2 243.7678} C_DIS
LIN {X -96.1615,Y -53.2501,Z 115,A -154.5997,B 24.9457,C -1.7029,E1 24.8606,E2 240.3784} C_DIS
LIN {X -94.5018,Y -56.1419,Z 115,A -152.8426,B 24.9459,C -1.6989,E1 24.8631,E2 238.6216} C_DIS
LIN {X -92.7744,Y -58.9544,Z 115,A -151.0836,B 24.9461,C -1.6959,E1 24.8657,E2 236.8609} C_DIS
LIN {X -90.1746,Y -62.857,Z 115,A -148.7103,B 24.9467,C -1.6869,E1 24.8694,E2 234.4972} C_DIS
LIN {X -88.6384,Y -65.0054,Z 115,A -146.5994,B 24.9451,C -1.7123,E1 24.873,E2 232.3154} C_DIS
LIN {X -85.7894,Y -68.7242,Z 115,A -144.7753,B 24.947,C -1.682,E1 24.876,E2 230.555} C_DIS
LIN {X -83.6812,Y -71.2735,Z 115,A -143.0791,B 24.9473,C -1.6769,E1 24.8791,E2 228.8632} C_DIS
LIN {X -81.0157,Y -74.2893,Z 115,A -140.964,B 24.9476,C -1.6729,E1 24.883,E2 226.7484} C_DIS
LIN {X -78.3944,Y -77.051,Z 115,A -138.9779,B 24.9478,C -1.6686,E1 24.8869,E2 224.7639} C_DIS
LIN {X -75.7988,Y -79.6079,Z 115,A -136.997,B 24.9478,C -1.6678,E1 24.8909,E2 222.7766} C_DIS
LIN {X -73.225,Y -81.979,Z 115,A -135.2769,B 24.9484,C -1.66,E1 24.8944,E2 221.068} C_DIS
LIN {X -70.377,Y -84.4367,Z 115,A -133.2591,B 24.9484,C -1.6585,E1 24.8987,E2 219.046} C_DIS
LIN {X -66.7625,Y -87.3235,Z 115,A -130.9238,B 24.9489,C -1.6511,E1 24.9038,E2 216.7199} C_DIS
LIN {X -59.9911,Y -92.1081,Z 115,A -126.5278,B 24.9492,C -1.6467,E1 24.9139,E2 212.3192} C_DIS
LIN {X -56.5185,Y -94.2791,Z 115,A -124.3553,B 24.9492,C -1.645,E1 24.9191,E2 210.144} C_DIS
LIN {X -53.3719,Y -96.0935,Z 115,A -122.4407,B 24.9494,C -1.6433,E1 24.9237,E2 208.228} C_DIS
LIN {X -50.1512,Y -97.8127,Z 115,A -120.6436,B 24.9498,C -1.6365,E1 24.9282,E2 206.442} C_DIS
LIN {X -47.2674,Y -99.239,Z 115,A -118.873,B 24.9498,C -1.6383,E1 24.9326,E2 204.6626} C_DIS
LIN {X -43.9791,Y -100.7388,Z 115,A -117.0136,B 24.9498,C -1.6352,E1 24.9374,E2 202.806} C_DIS
LIN {X -40.4802,Y -102.1954,Z 115,A -115.288,B 24.9506,C -1.623,E1 24.9418,E2 201.1056} C_DIS
LIN {X -36.9835,Y -103.5136,Z 115,A -112.9975,B 24.9499,C -1.6352,E1 24.9478,E2 198.7814} C_DIS
LIN {X -33.5647,Y -104.6706,Z 115,A -110.8967,B 24.9494,C -1.6428,E1 24.9535,E2 196.6588} C_DIS
LIN {X -28.741,Y -106.0963,Z 115,A -108.5747,B 24.9503,C -1.6286,E1 24.9596,E2 194.3666} C_DIS
LIN {X -25.0812,Y -107.0211,Z 115,A -106.5752,B 24.9503,C -1.6289,E1 24.9651,E2 192.3638} C_DIS
LIN {X -21.5451,Y -107.7896,Z 115,A -104.6977,B 24.9503,C -1.6277,E1 24.9702,E2 190.4869} C_DIS
LIN {X -17.9534,Y -108.4443,Z 115,A -102.7606,B 24.9503,C -1.6285,E1 24.9755,E2 188.546} C_DIS
LIN {X -13.5895,Y -109.0783,Z 115,A -100.3428,B 24.95,C -1.633,E1 24.9823,E2 186.1156} C_DIS
LIN {X -9.48,Y -109.5124,Z 115,A -98.2025,B 24.95,C -1.6322,E1 24.9882,E2 183.9761} C_DIS
LIN {X -5.4556,Y -109.7864,Z 115,A -96.3316,B 24.9507,C -1.6226,E1 24.9934,E2 182.1274} C_DIS
LIN {X -2.6407,Y -109.8902,Z 115,A -94.7147,B 24.9503,C -1.6291,E1 24.9979,E2 180.495} C_DIS
LIN {X 0.7808,Y -109.9135,Z 115,A -93.6591,B 24.9521,C -1.599,E1 25.0007,E2 179.5107} C_DIS
Enddeposition()
LIN {X 0.7808,Y -109.9135,Z 115,A -93.6591,B 24.9521,C -1.599,E1 25.0007,E2 179.5107} C_DIS
Startdeposition()
$VEL.CP = VEL_PRINT
LIN {X -1.0104,Y -109.003,Z 115,A -94.6962,B 24.9514,C -1.6108,E1 24.9979,E2 180.5197} C_DIS
LIN {X -3.6919,Y -108.9452,Z 115,A -96.1398,B 24.9514,C -1.6092,E1 24.9938,E2 181.9673} C_DIS
LIN {X -6.6909,Y -108.8036,Z 115,A -97.6824,B 24.9514,C -1.6106,E1 24.9895,E2 183.5072} C_DIS
LIN {X -9.3532,Y -108.6072,Z 115,A -99.0866,B 24.9514,C -1.6106,E1 24.9856,E2 184.9119} C_DIS
LIN {X -11.6323,Y -108.3851,Z 115,A -100.2992,B 24.9514,C -1.6103,E1 24.9822,E2 186.1257} C_DIS
LIN {X -14.679,Y -108.0163,Z 115,A -101.9033,B 24.9514,C -1.611,E1 24.9778,E2 187.7295} C_DIS
LIN {X -16.993,Y -107.675,Z 115,A -103.1669,B 24.9514,C -1.6099,E1 24.9743,E2 188.9968} C_DIS
LIN {X -19.6255,Y -107.2265,Z 115,A -104.6986,B 24.9517,C -1.6052,E1 24.9701,E2 190.5412} C_DIS
LIN {X -23.2401,Y -106.501,Z 115,A -106.5319,B 24.9514,C -1.6103,E1 24.9651,E2 192.3645} C_DIS
LIN {X -26.0833,Y -105.8408,Z 115,A -108.027,B 24.9513,C -1.6127,E1 24.961,E2 193.856} C_DIS
LIN {X -29.0749,Y -105.0603,Z 115,A -109.6418,B 24.9512,C -1.6141,E1 24.9567,E2 195.47} C_DIS
LIN {X -31.4942,Y -104.3597,Z 115,A -110.9579,B 24.9512,C -1.6153,E1 24.9531,E2 196.7853} C_DIS
LIN {X -33.8883,Y -103.6063,Z 115,A -112.3031,B 24.9512,C -1.6153,E1 24.9496,E2 198.1329} C_DIS
LIN {X -36.7217,Y -102.6378,Z 115,A -113.8658,B 24.951,C -1.6171,E1 24.9454,E2 199.6945} C_DIS
LIN {X -38.9314,Y -101.8186,Z 115,A -115.1073,B 24.951,C -1.6181,E1 24.9422,E2 200.936} C_DIS
LIN {X -41.4133,Y -100.8346,Z 115,A -116.5137,B 24.9509,C -1.6194,E1 24.9386,E2 202.3425} C_DIS
LIN {X -43.7397,Y -99.8471,Z 115,A -117.8674,B 24.9509,C -1.6198,E1 24.9351,E2 203.6984} C_DIS
LIN {X -46.6059,Y -98.5439,Z 115,A -119.5045,B 24.9507,C -1.6224,E1 24.9309,E2 205.3335} C_DIS
LIN {X -49.0058,Y -97.3726,Z 115,A -121.1059,B 24.951,C -1.6163,E1 24.9269,E2 206.9535} C_DIS
LIN {X -52.0756,Y -95.7638,Z 115,A -122.8219,B 24.9506,C -1.623,E1 24.9227,E2 208.6586} C_DIS
LIN {X -54.8952,Y -94.1781,Z 115,A -124.4416,B 24.9503,C -1.6285,E1 24.9188,E2 210.2699} C_DIS
LIN {X -57.1804,Y -92.8084,Z 115,A -125.9784,B 24.9505,C -1.6252,E1 24.9151,E2 211.8192} C_DIS
LIN {X -59.9861,Y -91.0177,Z 115,A -127.6993,B 24.9503,C -1.6291,E1 24.9111,E2 213.5364} C_DIS
LIN {X -62.5866,Y -89.2507,Z 115,A -129.2599,B 24.9499,C -1.6354,E1 24.9075,E2 215.0873} C_DIS
LIN {X -64.698,Y -87.7318,Z 115,A -130.8147,B 24.9502,C -1.6305,E1 24.9039,E2 216.6593} C_DIS
LIN {X -67.5679,Y -85.5403,Z 115,A -132.5488,B 24.9496,C -1.6403,E1 24.9002,E2 218.3764} C_DIS
LIN {X -69.6693,Y -83.8376,Z 115,A -133.968,B 24.9494,C -1.6431,E1 24.8971,E2 219.7944} C_DIS
LIN {X -71.7024,Y -82.1056,Z 115,A -135.4403,B 24.9494,C -1.6431,E1 24.894,E2 221.2722} C_DIS
LIN {X -74.154,Y -79.9007,Z 115,A -137.2991,B 24.9494,C -1.6418,E1 24.8901,E2 223.1419} C_DIS
LIN {X -76.6086,Y -77.5479,Z 115,A -138.9138,B 24.9488,C -1.6522,E1 24.8869,E2 224.7385} C_DIS
LIN {X -78.5839,Y -75.5457,Z 115,A -140.4532,B 24.9488,C -1.6531,E1 24.8839,E2 226.2824} C_DIS
LIN {X -80.6534,Y -73.3337,Z 115,A -141.9994,B 24.9485,C -1.6584,E1 24.881,E2 227.8228} C_DIS
LIN {X -82.5343,Y -71.2115,Z 115,A -143.6736,B 24.9487,C -1.6547,E1 24.8779,E2 229.5132} C_DIS
LIN {X -84.7628,Y -68.5408,Z 115,A -145.4299,B 24.9482,C -1.6618,E1 24.8748,E2 231.2607} C_DIS
LIN {X -87.5685,Y -64.921,Z 115,A -147.7506,B 24.9477,C -1.671,E1 24.8709,E2 233.5707} C_DIS
LIN {X -89.8821,Y -61.6782,Z 115,A -149.8586,B 24.9474,C -1.6757,E1 24.8675,E2 235.6778} C_DIS
LIN {X -91.1928,Y -59.7205,Z 115,A -151.1058,B 24.9472,C -1.6786,E1 24.8656,E2 236.9243} C_DIS
LIN {X -92.8048,Y -57.1863,Z 115,A -152.6935,B 24.947,C -1.6824,E1 24.8632,E2 238.5111} C_DIS
LIN {X -94.6797,Y -54.0224,Z 115,A -154.6385,B 24.9467,C -1.6872,E1 24.8605,E2 240.4548} C_DIS
LIN {X -96.0215,Y -51.6005,Z 115,A -156.1414,B 24.9465,C -1.6893,E1 24.8585,E2 241.9605} C_DIS
LIN {X -97.2305,Y -49.2842,Z 115,A -157.4811,B 24.9462,C -1.6944,E1 24.8568,E2 243.2952} C_DIS
LIN {X -98.3894,Y -46.9274,Z 115,A -158.8763,B 24.946,C -1.6978,E1 24.8551,E2 244.69} C_DIS
LIN {X -99.6586,Y -44.172,Z 115,A -160.4757,B 24.9457,C -1.7021,E1 24.8532,E2 246.2877} C_DIS
LIN {X -100.7107,Y -41.7177,Z 115,A -161.8898,B 24.9455,C -1.7058,E1 24.8517,E2 247.701} C_DIS
LIN {X -101.9521,Y -38.5789,Z 115,A -163.7326,B 24.9453,C -1.7085,E1 24.8498,E2 249.5477} C_DIS
LIN {X -102.8784,Y -36.036,Z 115,A -165.1575,B 24.945,C -1.7126,E1 24.8485,E2 250.9708} C_DIS
LIN {X -103.919,Y -32.9218,Z 115,A -166.8444,B 24.9446,C -1.7193,E1 24.847,E2 252.6515} C_DIS
LIN {X -104.5524,Y -30.8445,Z 115,A -168.063,B 24.9446,C -1.7199,E1 24.846,E2 253.8757} C_DIS
LIN {X -105.5457,Y -27.2523,Z 115,A -170.0798,B 24.9443,C -1.7237,E1 24.8446,E2 255.8951} C_DIS
LIN {X -106.3006,Y -24.1435,Z 115,A -171.6898,B 24.9438,C -1.7316,E1 24.8436,E2 257.4956} C_DIS
LIN {X -107.0979,Y -20.3148,Z 115,A -173.7598,B 24.9434,C -1.7375,E1 24.8424,E2 259.5638} C_DIS
LIN {X -107.5508,Y -17.7603,Z 115,A -175.1556,B 24.9432,C -1.7407,E1 24.8418,E2 260.9605} C_DIS
LIN {X -107.97,Y -15.0048,Z 115,A -176.5759,B 24.9428,C -1.747,E1 24.8412,E2 262.3742} C_DIS
LIN {X -108.3439,Y -12.0248,Z 115,A -178.1628,B 24.9425,C -1.7517,E1 24.8407,E2 263.9594} C_DIS
LIN {X -108.6078,Y -9.3462,Z 115,A -179.5867,B 24.9422,C -1.7559,E1 24.8403,E2 265.3818} C_DIS
LIN {X -108.7817,Y -7.0159,Z 115,A 179.1728,B 24.942,C -1.7594,E1 24.8401,E2 266.6214} C_DIS
LIN {X -108.9209,Y -4.3492,Z 115,A 177.7262,B 24.9418,C -1.7623,E1 24.8399,E2 268.0697} C_DIS
LIN {X -109.0008,Y -1.3469,Z 115,A 176.1603,B 24.9414,C -1.7679,E1 24.8398,E2 269.6318} C_DIS
LIN {X -109.0009,Y 1.3413,Z 115,A 174.748,B 24.9411,C -1.7725,E1 24.8398,E2 271.0416} C_DIS
LIN {X -108.9456,Y 3.6774,Z 115,A 173.4773,B 24.941,C -1.7749,E1 24.8399,E2 272.3141} C_DIS
LIN {X -108.8208,Y 6.3813,Z 115,A 172.0499,B 24.9407,C -1.7793,E1 24.8401,E2 273.7396} C_DIS
LIN {X -108.608,Y 9.3435,Z 115,A 170.5062,B 24.9403,C -1.785,E1 24.8405,E2 275.279} C_DIS
LIN {X -108.3465,Y 12.0007,Z 115,A 169.0951,B 24.94,C -1.7893,E1 24.8409,E2 276.6883} C_DIS
LIN {X -108.0167,Y 14.6765,Z 115,A 167.6468,B 24.9398,C -1.7927,E1 24.8414,E2 278.1371} C_DIS
LIN {X -107.6703,Y 17.0239,Z 115,A 166.3702,B 24.9396,C -1.7957,E1 24.8419,E2 279.4142} C_DIS
LIN {X -107.223,Y 19.6448,Z 115,A 164.9668,B 24.9393,C -1.8,E1 24.8426,E2 280.8157} C_DIS
LIN {X -106.6446,Y 22.5817,Z 115,A 163.4188,B 24.9389,C -1.806,E1 24.8435,E2 282.3586} C_DIS
LIN {X -106.0614,Y 25.179,Z 115,A 162.0074,B 24.9386,C -1.81,E1 24.8444,E2 283.7687} C_DIS
LIN {X -105.4977,Y 27.439,Z 115,A 160.7379,B 24.9384,C -1.8122,E1 24.8452,E2 285.0403} C_DIS
LIN {X -104.4521,Y 31.1825,Z 115,A 158.6934,B 24.938,C -1.8187,E1 24.8468,E2 287.0812} C_DIS
LIN {X -103.6088,Y 33.8806,Z 115,A 157.1899,B 24.9377,C -1.8227,E1 24.8481,E2 288.5838} C_DIS
LIN {X -102.638,Y 36.7213,Z 115,A 155.6329,B 24.9373,C -1.8284,E1 24.8495,E2 290.136} C_DIS
LIN {X -101.8261,Y 38.9115,Z 115,A 154.3973,B 24.9371,C -1.8319,E1 24.8507,E2 291.3702} C_DIS
LIN {X -100.8432,Y 41.3923,Z 115,A 152.985,B 24.9368,C -1.8359,E1 24.8522,E2 292.7809} C_DIS
LIN {X -99.667,Y 44.1528,Z 115,A 151.401,B 24.9365,C -1.8404,E1 24.854,E2 294.3629} C_DIS
LIN {X -97.9581,Y 47.8246,Z 115,A 149.2557,B 24.9361,C -1.8462,E1 24.8565,E2 296.506} C_DIS
LIN {X -96.7576,Y 50.2093,Z 115,A 147.8453,B 24.9358,C -1.8501,E1 24.8583,E2 297.9146} C_DIS
LIN {X -95.4988,Y 52.5641,Z 115,A 146.4303,B 24.9356,C -1.8538,E1 24.8602,E2 299.3283} C_DIS
LIN {X -94.2231,Y 54.817,Z 115,A 145.0414,B 24.9354,C -1.8568,E1 24.8621,E2 300.7174} C_DIS
LIN {X -92.791,Y 57.2084,Z 115,A 143.5988,B 24.935,C -1.8618,E1 24.8642,E2 302.1555} C_DIS
LIN {X -91.3656,Y 59.4585,Z 115,A 142.1843,B 24.9348,C -1.8652,E1 24.8663,E2 303.5689} C_DIS
LIN {X -90.0714,Y 61.3988,Z 115,A 140.9441,B 24.9346,C -1.8681,E1 24.8683,E2 304.8083} C_DIS
LIN {X -88.5435,Y 63.5824,Z 115,A 139.5215,B 24.9344,C -1.8712,E1 24.8706,E2 306.2306} C_DIS
LIN {X -86.8995,Y 65.812,Z 115,A 137.9597,B 24.9344,C -1.8712,E1 24.8732,E2 307.7999} C_DIS
LIN {X -84.6674,Y 68.6586,Z 115,A 136.1596,B 24.9337,C -1.88,E1 24.8763,E2 309.5874} C_DIS
LIN {X -82.9701,Y 70.7003,Z 115,A 134.7558,B 24.9335,C -1.8834,E1 24.8788,E2 310.9897} C_DIS
LIN {X -81.0936,Y 72.8452,Z 115,A 133.2582,B 24.9332,C -1.8872,E1 24.8816,E2 312.4849} C_DIS
LIN {X -79.3431,Y 74.7478,Z 115,A 131.8075,B 24.9332,C -1.8872,E1 24.8843,E2 313.9421} C_DIS
LIN {X -76.9293,Y 77.2312,Z 115,A 129.9085,B 24.9332,C -1.8886,E1 24.8881,E2 315.8457} C_DIS
LIN {X -74.3371,Y 79.7294,Z 115,A 128.0401,B 24.9327,C -1.894,E1 24.8919,E2 317.7089} C_DIS
LIN {X -71.673,Y 82.1313,Z 115,A 126.1721,B 24.9324,C -1.899,E1 24.8957,E2 319.5724} C_DIS
LIN {X -68.7475,Y 84.5953,Z 115,A 124.192,B 24.932,C -1.9047,E1 24.9,E2 321.5466} C_DIS
LIN {X -66.3976,Y 86.452,Z 115,A 122.5877,B 24.9318,C -1.9069,E1 24.9035,E2 323.1515} C_DIS
LIN {X -63.8632,Y 88.343,Z 115,A 120.9825,B 24.9314,C -1.9125,E1 24.9071,E2 324.749} C_DIS
LIN {X -61.6546,Y 89.8983,Z 115,A 119.5582,B 24.9312,C -1.9152,E1 24.9104,E2 326.1719} C_DIS
LIN {X -59.7139,Y 91.1972,Z 115,A 118.324,B 24.9311,C -1.9173,E1 24.9133,E2 327.4049} C_DIS
LIN {X -57.1812,Y 92.8079,Z 115,A 116.7418,B 24.9309,C -1.9201,E1 24.917,E2 328.9856} C_DIS
LIN {X -55.1788,Y 94.0105,Z 115,A 115.5074,B 24.9307,C -1.9221,E1 24.92,E2 330.219} C_DIS
LIN {X -52.8609,Y 95.3331,Z 115,A 114.0992,B 24.9306,C -1.9244,E1 24.9234,E2 331.6259} C_DIS
LIN {X -50.5317,Y 96.5878,Z 115,A 112.6978,B 24.9304,C -1.9263,E1 24.9268,E2 333.0266} C_DIS
LIN {X -48.1111,Y 97.8161,Z 115,A 111.3239,B 24.9301,C -1.9307,E1 24.9302,E2 334.3938} C_DIS
LIN {X -45.6936,Y 98.9685,Z 115,A 109.8134,B 24.9302,C -1.9289,E1 24.9341,E2 335.9124} C_DIS
LIN {X -43.2303,Y 100.0692,Z 115,A 108.4002,B 24.9301,C -1.9312,E1 24.9377,E2 337.3234} C_DIS
LIN {X -40.4652,Y 101.2203,Z 115,A 106.8598,B 24.9298,C -1.9347,E1 24.9417,E2 338.859} C_DIS
LIN {X -37.9793,Y 102.1792,Z 115,A 105.4532,B 24.9298,C -1.9363,E1 24.9453,E2 340.2646} C_DIS
LIN {X -35.732,Y 102.9851,Z 115,A 104.196,B 24.9296,C -1.9378,E1 24.9486,E2 341.5207} C_DIS
LIN {X -32.9083,Y 103.9232,Z 115,A 102.6327,B 24.9295,C -1.9397,E1 24.9528,E2 343.0824} C_DIS
LIN {X -29.0986,Y 105.0535,Z 115,A 100.5367,B 24.9293,C -1.9417,E1 24.9584,E2 345.1771} C_DIS
LIN {X -26.5414,Y 105.7284,Z 115,A 99.1532,B 24.9292,C -1.9433,E1 24.9621,E2 346.5587} C_DIS
LIN {X -24.1946,Y 106.2888,Z 115,A 97.8344,B 24.9292,C -1.9425,E1 24.9657,E2 347.8811} C_DIS
LIN {X -21.5846,Y 106.8494,Z 115,A 96.4633,B 24.9291,C -1.945,E1 24.9695,E2 349.2481} C_DIS
LIN {X -18.6332,Y 107.4049,Z 115,A 94.8832,B 24.929,C -1.9461,E1 24.9738,E2 350.8271} C_DIS
LIN {X -15.9968,Y 107.8291,Z 115,A 93.4765,B 24.929,C -1.9469,E1 24.9777,E2 352.233} C_DIS
LIN {X -12.0002,Y 108.3466,Z 115,A 91.3623,B 24.9288,C -1.9484,E1 24.9835,E2 354.3454} C_DIS
LIN {X -9.344,Y 108.608,Z 115,A 89.9546,B 24.9288,C -1.9489,E1 24.9875,E2 355.7526} C_DIS
LIN {X -7.0143,Y 108.7818,Z 115,A 88.7218,B 24.9288,C -1.9492,E1 24.9909,E2 356.9851} C_DIS
LIN {X -4.3485,Y 108.9209,Z 115,A 87.3082,B 24.9288,C -1.9492,E1 24.9948,E2 358.3988} C_DIS
LIN {X -1.3336,Y 109.001,Z 115,A 85.7332,B 24.9288,C -1.9501,E1 24.9992,E2 359.972} C_DIS
LIN {X 2.3485,Y 108.9824,Z 115,A 83.7955,B 24.9287,C -1.9503,E1 25.0046,E2 361.909} C_DIS
LIN {X 5.3496,Y 108.8779,Z 115,A 82.217,B 24.9287,C -1.9503,E1 25.009,E2 363.4868} C_DIS
LIN {X 8.0148,Y 108.7141,Z 115,A 80.8144,B 24.9287,C -1.9503,E1 25.0129,E2 364.8888} C_DIS
LIN {X 12.0211,Y 108.3443,Z 115,A 78.7016,B 24.9287,C -1.9502,E1 25.0188,E2 367.0007} C_DIS
LIN {X 14.6742,Y 108.017,Z 115,A 77.2956,B 24.9287,C -1.9498,E1 25.0227,E2 368.4064} C_DIS
LIN {X 16.9863,Y 107.6761,Z 115,A 76.035,B 24.9288,C -1.9482,E1 25.0262,E2 369.6698} C_DIS
LIN {X 20.6549,Y 107.0324,Z 115,A 74.0675,B 24.9289,C -1.947,E1 25.0316,E2 371.6378} C_DIS
LIN {X 23.5624,Y 106.4307,Z 115,A 72.52,B 24.9289,C -1.9468,E1 25.0358,E2 373.1839} C_DIS
LIN {X 26.4853,Y 105.7428,Z 115,A 70.9756,B 24.9289,C -1.9473,E1 25.04,E2 374.725} C_DIS
LIN {X 29.0956,Y 105.0544,Z 115,A 69.5687,B 24.9289,C -1.9468,E1 25.0438,E2 376.1306} C_DIS
LIN {X 31.6518,Y 104.3128,Z 115,A 68.1658,B 24.929,C -1.9456,E1 25.0476,E2 377.534} C_DIS
LIN {X 33.8737,Y 103.611,Z 115,A 66.9072,B 24.9292,C -1.9433,E1 25.0509,E2 378.7957} C_DIS
LIN {X 36.7368,Y 102.6323,Z 115,A 65.353,B 24.9292,C -1.9433,E1 25.055,E2 380.3467} C_DIS
LIN {X 38.9278,Y 101.82,Z 115,A 64.126,B 24.9292,C -1.9423,E1 25.0582,E2 381.5736} C_DIS
LIN {X 41.4099,Y 100.836,Z 115,A 62.7257,B 24.9294,C -1.9409,E1 25.0618,E2 382.9739} C_DIS
LIN {X 44.1728,Y 99.6583,Z 115,A 61.151,B 24.9294,C -1.9393,E1 25.0659,E2 384.5487} C_DIS
LIN {X 46.6005,Y 98.5464,Z 115,A 59.6214,B 24.93,C -1.9324,E1 25.0698,E2 386.0907} C_DIS
LIN {X 49.5926,Y 97.0728,Z 115,A 57.946,B 24.93,C -1.9334,E1 25.0739,E2 387.7591} C_DIS
LIN {X 52.5673,Y 95.497,Z 115,A 56.2409,B 24.93,C -1.9337,E1 25.0781,E2 389.4588} C_DIS
LIN {X 54.896,Y 94.1777,Z 115,A 54.837,B 24.93,C -1.9318,E1 25.0815,E2 390.8629} C_DIS
LIN {X 58.0361,Y 92.2739,Z 115,A 52.8803,B 24.9303,C -1.9277,E1 25.0862,E2 392.823} C_DIS
LIN {X 60.5571,Y 90.6413,Z 115,A 51.3397,B 24.9304,C -1.9268,E1 25.0898,E2 394.3608} C_DIS
LIN {X 62.4854,Y 89.321,Z 115,A 50.1151,B 24.9305,C -1.9249,E1 25.0926,E2 395.5857} C_DIS
LIN {X 64.6754,Y 87.7484,Z 115,A 48.7034,B 24.9307,C -1.9226,E1 25.0958,E2 396.9977} C_DIS
LIN {X 66.9353,Y 86.0377,Z 115,A 47.2192,B 24.9309,C -1.9201,E1 25.0991,E2 398.4823} C_DIS
LIN {X 69.1504,Y 84.2687,Z 115,A 45.5487,B 24.9316,C -1.9097,E1 25.1027,E2 400.1714} C_DIS
LIN {X 71.8311,Y 81.9932,Z 115,A 43.8449,B 24.9315,C -1.9122,E1 25.1063,E2 401.8625} C_DIS
LIN {X 74.199,Y 79.8592,Z 115,A 42.0552,B 24.932,C -1.9039,E1 25.11,E2 403.6646} C_DIS
LIN {X 76.6042,Y 77.5523,Z 115,A 40.4831,B 24.9318,C -1.9079,E1 25.1131,E2 405.2207} C_DIS
LIN {X 78.4812,Y 75.6523,Z 115,A 39.0861,B 24.932,C -1.9051,E1 25.1158,E2 406.6183} C_DIS
LIN {X 80.3201,Y 73.697,Z 115,A 37.6818,B 24.9322,C -1.9022,E1 25.1185,E2 408.0232} C_DIS
LIN {X 82.194,Y 71.6012,Z 115,A 36.1367,B 24.9326,C -1.8959,E1 25.1214,E2 409.5762} C_DIS
LIN {X 84.5817,Y 68.7643,Z 115,A 34.2284,B 24.9328,C -1.8931,E1 25.1248,E2 411.4826} C_DIS
LIN {X 86.3419,Y 66.5404,Z 115,A 32.7424,B 24.9331,C -1.8896,E1 25.1273,E2 412.9696} C_DIS
LIN {X 88.354,Y 63.848,Z 115,A 31.0328,B 24.9332,C -1.8877,E1 25.1302,E2 414.6757} C_DIS
LIN {X 89.8913,Y 61.6648,Z 115,A 29.638,B 24.9334,C -1.8845,E1 25.1324,E2 416.0711} C_DIS
LIN {X 91.1914,Y 59.7227,Z 115,A 28.4144,B 24.9336,C -1.8815,E1 25.1343,E2 417.2957} C_DIS
LIN {X 92.8035,Y 57.1884,Z 115,A 26.845,B 24.9339,C -1.8777,E1 25.1366,E2 418.8661} C_DIS
LIN {X 94.0128,Y 55.1748,Z 115,A 25.6179,B 24.9341,C -1.8747,E1 25.1384,E2 420.0938} C_DIS
LIN {X 95.3313,Y 52.864,Z 115,A 24.2277,B 24.9344,C -1.8713,E1 25.1403,E2 421.485} C_DIS
LIN {X 96.567,Y 50.5711,Z 115,A 22.8755,B 24.9346,C -1.8682,E1 25.142,E2 422.8373} C_DIS
LIN {X 97.8192,Y 48.105,Z 115,A 21.4211,B 24.9349,C -1.8641,E1 25.1439,E2 424.2937} C_DIS
LIN {X 98.968,Y 45.6947,Z 115,A 19.9948,B 24.9352,C -1.8591,E1 25.1456,E2 425.7241} C_DIS
LIN {X 100.0576,Y 43.2569,Z 115,A 18.5995,B 24.9355,C -1.8554,E1 25.1471,E2 427.1205} C_DIS
LIN {X 101.2277,Y 40.4465,Z 115,A 17.0447,B 24.9357,C -1.8527,E1 25.1488,E2 428.6732} C_DIS
LIN {X 102.1845,Y 37.9646,Z 115,A 15.6603,B 24.9359,C -1.8491,E1 25.1501,E2 430.0582} C_DIS
LIN {X 102.9711,Y 35.7719,Z 115,A 14.436,B 24.9362,C -1.8455,E1 25.1513,E2 431.2842} C_DIS
LIN {X 103.9161,Y 32.931,Z 115,A 12.8717,B 24.9365,C -1.8411,E1 25.1526,E2 432.8499} C_DIS
LIN {X 104.5944,Y 30.703,Z 115,A 11.6361,B 24.9368,C -1.8369,E1 25.1536,E2 434.0884} C_DIS
LIN {X 105.322,Y 28.1062,Z 115,A 10.2159,B 24.9371,C -1.8324,E1 25.1547,E2 435.511} C_DIS
LIN {X 106.1741,Y 24.691,Z 115,A 8.3409,B 24.9375,C -1.8256,E1 25.1559,E2 437.3913} C_DIS
LIN {X 106.8032,Y 21.8094,Z 115,A 6.8328,B 24.9377,C -1.8226,E1 25.1568,E2 438.8977} C_DIS
LIN {X 107.404,Y 18.6382,Z 115,A 5.1852,B 24.938,C -1.8194,E1 25.1576,E2 440.5433} C_DIS
LIN {X 107.8283,Y 16.0019,Z 115,A 3.6343,B 24.9387,C -1.8084,E1 25.1583,E2 442.1109} C_DIS
LIN {X 108.2753,Y 12.6106,Z 115,A 1.9572,B 24.9387,C -1.808,E1 25.1588,E2 443.779} C_DIS
LIN {X 108.6074,Y 9.351,Z 115,A 0.2959,B 24.9389,C -1.8051,E1 25.1593,E2 445.4373} C_DIS
LIN {X 108.7814,Y 7.0206,Z 115,A -0.9248,B 24.9392,C -1.8015,E1 25.1595,E2 446.6592} C_DIS
LIN {X 108.9207,Y 4.3542,Z 115,A -2.352,B 24.9395,C -1.7959,E1 25.1597,E2 448.0911} C_DIS
LIN {X 108.9972,Y 1.5425,Z 115,A -3.7826,B 24.9397,C -1.7932,E1 25.1597,E2 449.5195} C_DIS
LIN {X 109.0017,Y -1.2452,Z 115,A -5.2378,B 24.94,C -1.7889,E1 25.1597,E2 450.9763} C_DIS
LIN {X 108.9456,Y -3.6783,Z 115,A -6.5436,B 24.9404,C -1.7836,E1 25.1597,E2 452.2868} C_DIS
LIN {X 108.8045,Y -6.6766,Z 115,A -8.0788,B 24.9406,C -1.7803,E1 25.1594,E2 453.8207} C_DIS
LIN {X 108.6067,Y -9.3586,Z 115,A -9.4795,B 24.9409,C -1.7763,E1 25.1591,E2 455.2226} C_DIS
LIN {X 108.3449,Y -12.016,Z 115,A -10.8758,B 24.9411,C -1.772,E1 25.1587,E2 456.6206} C_DIS
LIN {X 108.0177,Y -14.6693,Z 115,A -12.2715,B 24.9414,C -1.7679,E1 25.1582,E2 458.018} C_DIS
LIN {X 107.6768,Y -16.9815,Z 115,A -13.5235,B 24.9418,C -1.7629,E1 25.1577,E2 459.2743} C_DIS
LIN {X 107.1067,Y -20.2689,Z 115,A -15.3187,B 24.9423,C -1.7554,E1 25.1568,E2 461.0768} C_DIS
LIN {X 106.4793,Y -23.3394,Z 115,A -16.9473,B 24.9425,C -1.7509,E1 25.1558,E2 462.7064} C_DIS
LIN {X 105.7428,Y -26.4853,Z 115,A -18.5551,B 24.9426,C -1.7494,E1 25.1548,E2 464.3084} C_DIS
LIN {X 105.0623,Y -29.0674,Z 115,A -19.9483,B 24.9429,C -1.7454,E1 25.1538,E2 465.7031} C_DIS
LIN {X 104.3039,Y -31.6807,Z 115,A -21.3513,B 24.9431,C -1.742,E1 25.1527,E2 467.106} C_DIS
LIN {X 103.6051,Y -33.8921,Z 115,A -22.5955,B 24.9434,C -1.7371,E1 25.1516,E2 468.3548} C_DIS
LIN {X 102.7973,Y -36.2672,Z 115,A -23.9302,B 24.9438,C -1.7322,E1 25.1504,E2 469.6934} C_DIS
LIN {X 101.8196,Y -38.9288,Z 115,A -25.3705,B 24.9439,C -1.7298,E1 25.149,E2 471.1315} C_DIS
LIN {X 100.8356,Y -41.4108,Z 115,A -26.7647,B 24.9442,C -1.7259,E1 25.1475,E2 472.5272} C_DIS
LIN {X 99.6579,Y -44.1737,Z 115,A -28.3329,B 24.9445,C -1.7214,E1 25.1458,E2 474.0973} C_DIS
LIN {X 98.545,Y -46.6035,Z 115,A -29.7446,B 24.9448,C -1.7169,E1 25.1441,E2 475.5121} C_DIS
LIN {X 97.3576,Y -49.0355,Z 115,A -31.1386,B 24.945,C -1.7138,E1 25.1424,E2 476.9059} C_DIS
LIN {X 96.2861,Y -51.1044,Z 115,A -32.3912,B 24.9453,C -1.709,E1 25.1407,E2 478.1632} C_DIS
LIN {X 94.8471,Y -53.7312,Z 115,A -33.9227,B 24.9454,C -1.7062,E1 25.1387,E2 479.6934} C_DIS
LIN {X 93.5061,Y -56.0321,Z 115,A -35.3142,B 24.9457,C -1.7025,E1 25.1367,E2 481.0864} C_DIS
LIN {X 92.2859,Y -58.017,Z 115,A -36.5645,B 24.946,C -1.6979,E1 25.1348,E2 482.3413} C_DIS
LIN {X 90.6599,Y -60.5289,Z 115,A -38.0881,B 24.9461,C -1.6955,E1 25.1325,E2 483.8628} C_DIS
LIN {X 89.348,Y -62.4465,Z 115,A -39.2905,B 24.9463,C -1.6929,E1 25.1306,E2 485.0654} C_DIS
LIN {X 87.5511,Y -64.9446,Z 115,A -41.0874,B 24.9471,C -1.6806,E1 25.1276,E2 486.8828} C_DIS
LIN {X 85.5208,Y -67.5925,Z 115,A -42.6595,B 24.9469,C -1.6838,E1 25.1249,E2 488.4398} C_DIS
LIN {X 83.8389,Y -69.6678,Z 115,A -44.0556,B 24.9471,C -1.6805,E1 25.1224,E2 489.8375} C_DIS
LIN {X 82.1066,Y -71.7012,Z 115,A -45.4534,B 24.9473,C -1.6771,E1 25.1199,E2 491.2369} C_DIS
LIN {X 80.1695,Y -73.8611,Z 115,A -47.0065,B 24.9476,C -1.6719,E1 25.117,E2 492.7952} C_DIS
LIN {X 78.1358,Y -76.0106,Z 115,A -48.5157,B 24.9477,C -1.67,E1 25.1141,E2 494.3025} C_DIS
LIN {X 76.2503,Y -77.9018,Z 115,A -49.9209,B 24.948,C -1.6665,E1 25.1113,E2 495.71} C_DIS
LIN {X 73.8165,Y -80.2104,Z 115,A -51.7376,B 24.9484,C -1.66,E1 25.1075,E2 497.5347} C_DIS
LIN {X 71.324,Y -82.436,Z 115,A -53.4236,B 24.9484,C -1.659,E1 25.104,E2 499.2164} C_DIS
LIN {X 68.7657,Y -84.5805,Z 115,A -55.2041,B 24.9487,C -1.6539,E1 25.1002,E2 501.002} C_DIS
LIN {X 66.4084,Y -86.4437,Z 115,A -56.7978,B 24.949,C -1.6499,E1 25.0967,E2 502.5994} C_DIS
LIN {X 63.1892,Y -88.824,Z 115,A -58.92,B 24.9493,C -1.6447,E1 25.0919,E2 504.7264} C_DIS
LIN {X 60.5492,Y -90.6465,Z 115,A -60.4984,B 24.9493,C -1.6459,E1 25.0882,E2 506.2966} C_DIS
LIN {X 58.5723,Y -91.9346,Z 115,A -61.7772,B 24.9495,C -1.6418,E1 25.0852,E2 507.5808} C_DIS
LIN {X 56.3133,Y -93.3354,Z 115,A -63.1317,B 24.9495,C -1.641,E1 25.082,E2 508.9329} C_DIS
LIN {X 54.019,Y -94.6817,Z 115,A -64.5242,B 24.9497,C -1.6387,E1 25.0786,E2 510.3267} C_DIS
LIN {X 51.6923,Y -95.9717,Z 115,A -65.9585,B 24.9499,C -1.6347,E1 25.0751,E2 511.7663} C_DIS
LIN {X 49.299,Y -97.2229,Z 115,A -67.3324,B 24.9499,C -1.6342,E1 25.0717,E2 513.1375} C_DIS
LIN {X 46.9031,Y -98.4011,Z 115,A -68.7308,B 24.9501,C -1.6322,E1 25.0682,E2 514.5371} C_DIS
LIN {X 44.175,Y -99.6573,Z 115,A -70.3118,B 24.9502,C -1.6296,E1 25.0642,E2 516.1203} C_DIS
LIN {X 41.5555,Y -100.7767,Z 115,A -71.7737,B 24.9502,C -1.6289,E1 25.0604,E2 517.5804} C_DIS
LIN {X 39.1557,Y -101.7336,Z 115,A -73.1373,B 24.9504,C -1.6268,E1 25.0568,E2 518.946} C_DIS
LIN {X 37.006,Y -102.5342,Z 115,A -74.3505,B 24.9505,C -1.6248,E1 25.0537,E2 520.1612} C_DIS
LIN {X 34.5239,Y -103.3961,Z 115,A -75.7611,B 24.9507,C -1.6218,E1 25.0499,E2 521.5762} C_DIS
LIN {X 31.6355,Y -104.3178,Z 115,A -77.3157,B 24.9507,C -1.6216,E1 25.0458,E2 523.1286} C_DIS
LIN {X 29.071,Y -105.0613,Z 115,A -78.7186,B 24.9508,C -1.62,E1 25.042,E2 524.5327} C_DIS
LIN {X 26.4864,Y -105.7425,Z 115,A -80.1216,B 24.9509,C -1.6187,E1 25.0382,E2 525.9368} C_DIS
LIN {X 23.5616,Y -106.4309,Z 115,A -81.7885,B 24.9512,C -1.6135,E1 25.0336,E2 527.6136} C_DIS
LIN {X 20.2658,Y -107.1073,Z 115,A -83.4988,B 24.9512,C -1.6144,E1 25.029,E2 529.3198} C_DIS
LIN {X 17.6372,Y -107.5714,Z 115,A -84.8965,B 24.9512,C -1.6136,E1 25.0251,E2 530.718} C_DIS
LIN {X 14.9976,Y -107.9711,Z 115,A -86.2646,B 24.9512,C -1.614,E1 25.0214,E2 532.0837} C_DIS
LIN {X 12.4745,Y -108.2912,Z 115,A -87.6231,B 24.9512,C -1.6123,E1 25.0176,E2 533.4453} C_DIS
LIN {X 9.3323,Y -108.6089,Z 115,A -89.2485,B 24.9512,C -1.6128,E1 25.0131,E2 535.0686} C_DIS
LIN {X 7.0046,Y -108.7824,Z 115,A -90.4834,B 24.9513,C -1.612,E1 25.0096,E2 536.305} C_DIS
LIN {X 4.341,Y -108.9212,Z 115,A -91.9158,B 24.9514,C -1.6102,E1 25.0056,E2 537.7411} C_DIS
LIN {X 0.7752,Y -109.0044,Z 115,A -93.4858,B 24.9507,C -1.6222,E1 25.0013,E2 539.2823} C_DIS
Enddeposition()
LIN {X 0.8075,Y -115.1575,Z 116,A -93.2729,B 24.9561,C -1.531,E1 25.0013,E2 539.2856} C_DIS
Startdeposition()
$VEL.CP = VEL_PRINT
LIN {X 2.9016,Y -115.1254,Z 116,A -91.9023,B 24.9552,C -1.5459,E1 25.0052,E2 537.88} C_DIS
LIN {X 5.7261,Y -115.0195,Z 116,A -90.4971,B 24.9552,C -1.5463,E1 25.0091,E2 536.4741} C_DIS
LIN {X 8.5471,Y -114.8444,Z 116,A -89.0922,B 24.9552,C -1.5469,E1 25.0131,E2 535.0684} C_DIS
LIN {X 11.2879,Y -114.6079,Z 116,A -87.6908,B 24.955,C -1.5491,E1 25.017,E2 533.6627} C_DIS
LIN {X 14.5615,Y -114.2362,Z 116,A -86.2647,B 24.9555,C -1.5406,E1 25.0209,E2 532.2578} C_DIS
LIN {X 16.9724,Y -113.9044,Z 116,A -84.8791,B 24.955,C -1.5492,E1 25.0248,E2 530.8529} C_DIS
LIN {X 20.2239,Y -113.3706,Z 116,A -83.4531,B 24.9555,C -1.5409,E1 25.0286,E2 529.4481} C_DIS
LIN {X 22.541,Y -112.9344,Z 116,A -82.0714,B 24.9549,C -1.5513,E1 25.0325,E2 528.0435} C_DIS
LIN {X 25.2322,Y -112.3642,Z 116,A -80.5045,B 24.9543,C -1.5615,E1 25.0368,E2 526.4545} C_DIS
LIN {X 28.0552,Y -111.6924,Z 116,A -79.2308,B 24.9547,C -1.5553,E1 25.0402,E2 525.1974} C_DIS
LIN {X 30.7879,Y -110.9702,Z 116,A -77.8276,B 24.9547,C -1.5566,E1 25.044,E2 523.7932} C_DIS
LIN {X 33.5019,Y -110.1812,Z 116,A -76.4247,B 24.9545,C -1.5581,E1 25.0478,E2 522.3893} C_DIS
LIN {X 36.1243,Y -109.35,Z 116,A -75.0596,B 24.9545,C -1.5596,E1 25.0514,E2 521.0232} C_DIS
LIN {X 38.8679,Y -108.4046,Z 116,A -73.6198,B 24.9543,C -1.5613,E1 25.0552,E2 519.5823} C_DIS
LIN {X 41.4464,Y -107.4457,Z 116,A -72.2552,B 24.9543,C -1.563,E1 25.0587,E2 518.2166} C_DIS
LIN {X 44.0707,Y -106.3962,Z 116,A -70.8534,B 24.9541,C -1.5648,E1 25.0624,E2 516.8138} C_DIS
LIN {X 46.7373,Y -105.2516,Z 116,A -69.4141,B 24.9541,C -1.5668,E1 25.0661,E2 515.3733} C_DIS
LIN {X 49.2383,Y -104.1056,Z 116,A -68.0501,B 24.9539,C -1.5688,E1 25.0695,E2 514.0081} C_DIS
LIN {X 51.7783,Y -102.8659,Z 116,A -66.6486,B 24.9538,C -1.5709,E1 25.073,E2 512.6054} C_DIS
LIN {X 54.3535,Y -101.5282,Z 116,A -65.1011,B 24.9533,C -1.5782,E1 25.0769,E2 511.045} C_DIS
LIN {X 56.7633,Y -100.2013,Z 116,A -63.8147,B 24.9534,C -1.5768,E1 25.08,E2 509.7656} C_DIS
LIN {X 59.2698,Y -98.7389,Z 116,A -62.4428,B 24.9534,C -1.5762,E1 25.0833,E2 508.3994} C_DIS
LIN {X 61.7353,Y -97.216,Z 116,A -61.0031,B 24.9533,C -1.5788,E1 25.0867,E2 506.9579} C_DIS
LIN {X 63.9808,Y -95.754,Z 116,A -59.6133,B 24.953,C -1.5841,E1 25.0899,E2 505.5604} C_DIS
LIN {X 66.3115,Y -94.155,Z 116,A -58.2131,B 24.9528,C -1.5867,E1 25.0932,E2 504.1589} C_DIS
LIN {X 68.6625,Y -92.454,Z 116,A -56.8083,B 24.9528,C -1.588,E1 25.0963,E2 502.7561} C_DIS
LIN {X 70.8516,Y -90.7879,Z 116,A -55.4136,B 24.9525,C -1.5921,E1 25.0994,E2 501.3566} C_DIS
LIN {X 73.3393,Y -88.7882,Z 116,A -54.0292,B 24.9529,C -1.5862,E1 25.1024,E2 499.9914} C_DIS
LIN {X 75.221,Y -87.202,Z 116,A -52.4729,B 24.9518,C -1.6045,E1 25.1058,E2 498.3981} C_DIS
LIN {X 77.4929,Y -85.1879,Z 116,A -51.2006,B 24.9522,C -1.5969,E1 25.1083,E2 497.1487} C_DIS
LIN {X 79.4092,Y -83.406,Z 116,A -49.8484,B 24.9519,C -1.6024,E1 25.1111,E2 495.7893} C_DIS
LIN {X 81.6097,Y -81.2523,Z 116,A -48.3993,B 24.9519,C -1.6023,E1 25.114,E2 494.3464} C_DIS
LIN {X 83.406,Y -79.4092,Z 116,A -47.0508,B 24.9515,C -1.6086,E1 25.1166,E2 492.9888} C_DIS
LIN {X 85.38,Y -77.2821,Z 116,A -45.615,B 24.9513,C -1.612,E1 25.1193,E2 491.5514} C_DIS
LIN {X 87.2509,Y -75.1635,Z 116,A -44.2505,B 24.9513,C -1.6137,E1 25.1218,E2 490.1891} C_DIS
LIN {X 89.0217,Y -73.0583,Z 116,A -42.8235,B 24.9508,C -1.62,E1 25.1244,E2 488.7536} C_DIS
LIN {X 90.7879,Y -70.8516,Z 116,A -41.4574,B 24.9508,C -1.6219,E1 25.1267,E2 487.3894} C_DIS
LIN {X 92.4993,Y -68.6022,Z 116,A -40.0274,B 24.9504,C -1.6269,E1 25.1291,E2 485.9546} C_DIS
LIN {X 94.155,Y -66.3115,Z 116,A -38.5166,B 24.9499,C -1.6358,E1 25.1316,E2 484.4302} C_DIS
LIN {X 95.754,Y -63.9808,Z 116,A -37.2635,B 24.9501,C -1.6325,E1 25.1335,E2 483.191} C_DIS
LIN {X 97.4789,Y -61.3178,Z 116,A -35.8497,B 24.9503,C -1.6293,E1 25.1356,E2 481.7919} C_DIS
LIN {X 98.7781,Y -59.2053,Z 116,A -34.4364,B 24.9495,C -1.6413,E1 25.1377,E2 480.3575} C_DIS
LIN {X 100.2381,Y -56.6975,Z 116,A -33.0674,B 24.9495,C -1.642,E1 25.1396,E2 478.9939} C_DIS
LIN {X 101.5993,Y -54.2204,Z 116,A -31.6364,B 24.9491,C -1.6474,E1 25.1415,E2 477.5578} C_DIS
LIN {X 102.8994,Y -51.7107,Z 116,A -30.2391,B 24.9489,C -1.6512,E1 25.1433,E2 476.1589} C_DIS
LIN {X 104.1056,Y -49.2383,Z 116,A -28.8791,B 24.9487,C -1.6549,E1 25.1449,E2 474.7975} C_DIS
LIN {X 105.3996,Y -46.4001,Z 116,A -27.4286,B 24.9487,C -1.6549,E1 25.1466,E2 473.3549} C_DIS
LIN {X 106.4246,Y -44.0009,Z 116,A -26.048,B 24.9482,C -1.6628,E1 25.1481,E2 471.9632} C_DIS
LIN {X 107.4457,Y -41.4464,Z 116,A -24.6882,B 24.948,C -1.6666,E1 25.1495,E2 470.602} C_DIS
LIN {X 108.4555,Y -38.7259,Z 116,A -23.1996,B 24.9475,C -1.6733,E1 25.1509,E2 469.1059} C_DIS
LIN {X 109.35,Y -36.1243,Z 116,A -21.8944,B 24.9475,C -1.6746,E1 25.1521,E2 467.805} C_DIS
LIN {X 110.2036,Y -33.4299,Z 116,A -20.4979,B 24.9472,C -1.6786,E1 25.1532,E2 466.4071} C_DIS
LIN {X 110.9908,Y -30.7153,Z 116,A -19.1013,B 24.9469,C -1.6826,E1 25.1543,E2 465.0089} C_DIS
LIN {X 111.8145,Y -27.5586,Z 116,A -17.6391,B 24.9471,C -1.6802,E1 25.1553,E2 463.5609} C_DIS
LIN {X 112.3803,Y -25.1585,Z 116,A -16.3046,B 24.9465,C -1.6892,E1 25.1561,E2 462.2127} C_DIS
LIN {X 112.9638,Y -22.393,Z 116,A -14.9114,B 24.9463,C -1.6932,E1 25.1569,E2 460.8184} C_DIS
LIN {X 113.4794,Y -19.614,Z 116,A -13.5114,B 24.946,C -1.6974,E1 25.1576,E2 459.4166} C_DIS
LIN {X 113.9266,Y -16.8232,Z 116,A -11.9399,B 24.9452,C -1.7099,E1 25.1583,E2 457.825} C_DIS
LIN {X 114.3051,Y -14.0222,Z 116,A -10.6848,B 24.9454,C -1.7073,E1 25.1587,E2 456.5835} C_DIS
LIN {X 114.6148,Y -11.2128,Z 116,A -9.3221,B 24.9452,C -1.7098,E1 25.1591,E2 455.2229} C_DIS
LIN {X 114.8555,Y -8.3966,Z 116,A -7.9256,B 24.945,C -1.7139,E1 25.1594,E2 453.825} C_DIS
LIN {X 115.0269,Y -5.5754,Z 116,A -6.5289,B 24.9447,C -1.718,E1 25.1596,E2 452.4269} C_DIS
LIN {X 115.1291,Y -2.7508,Z 116,A -5.1326,B 24.9444,C -1.7221,E1 25.1598,E2 451.0291} C_DIS
LIN {X 115.1613,Y 0,Z 116,A -3.7801,B 24.9442,C -1.7259,E1 25.1598,E2 449.6759} C_DIS
LIN {X 115.1254,Y 2.9016,Z 116,A -2.3397,B 24.9439,C -1.7304,E1 25.1598,E2 448.2335} C_DIS
LIN {X 115.0195,Y 5.7261,Z 116,A -0.9431,B 24.9436,C -1.7345,E1 25.1595,E2 446.8355} C_DIS
LIN {X 114.8444,Y 8.5471,Z 116,A 0.4873,B 24.9432,C -1.7402,E1 25.1593,E2 445.4002} C_DIS
LIN {X 114.6,Y 11.3629,Z 116,A 1.884,B 24.943,C -1.7442,E1 25.1589,E2 444.0021} C_DIS
LIN {X 114.2866,Y 14.1719,Z 116,A 3.2467,B 24.9428,C -1.7467,E1 25.1585,E2 442.6416} C_DIS
LIN {X 113.9044,Y 16.9724,Z 116,A 4.6433,B 24.9426,C -1.7507,E1 25.1579,E2 441.2438} C_DIS
LIN {X 113.3951,Y 20.0877,Z 116,A 6.0556,B 24.9427,C -1.7483,E1 25.1573,E2 439.8456} C_DIS
LIN {X 112.9496,Y 22.4671,Z 116,A 7.4334,B 24.9419,C -1.7602,E1 25.1565,E2 438.4476} C_DIS
LIN {X 112.3472,Y 25.3057,Z 116,A 8.8335,B 24.9418,C -1.7627,E1 25.1557,E2 437.0499} C_DIS
LIN {X 111.7111,Y 27.9822,Z 116,A 10.3637,B 24.941,C -1.7746,E1 25.1547,E2 435.5006} C_DIS
LIN {X 110.9702,Y 30.7879,Z 116,A 11.7833,B 24.9408,C -1.7779,E1 25.1536,E2 434.0813} C_DIS
LIN {X 110.1812,Y 33.5019,Z 116,A 13.0247,B 24.941,C -1.7744,E1 25.1526,E2 432.8551} C_DIS
LIN {X 109.2373,Y 36.4585,Z 116,A 14.4349,B 24.941,C -1.7728,E1 25.1514,E2 431.4567} C_DIS
LIN {X 108.4046,Y 38.8679,Z 116,A 15.853,B 24.9404,C -1.7836,E1 25.1501,E2 430.021} C_DIS
LIN {X 107.4181,Y 41.5166,Z 116,A 17.2502,B 24.9401,C -1.7874,E1 25.1487,E2 428.6228} C_DIS
LIN {X 106.3669,Y 44.1403,Z 116,A 18.6139,B 24.94,C -1.7895,E1 25.1473,E2 427.2615} C_DIS
LIN {X 105.103,Y 47.0672,Z 116,A 20.2558,B 24.9395,C -1.7967,E1 25.1454,E2 425.6116} C_DIS
LIN {X 104.0729,Y 49.3063,Z 116,A 21.4092,B 24.9395,C -1.7968,E1 25.1441,E2 424.4642} C_DIS
LIN {X 102.8659,Y 51.7783,Z 116,A 22.8357,B 24.939,C -1.8034,E1 25.1423,E2 423.0299} C_DIS
LIN {X 101.5642,Y 54.2872,Z 116,A 24.2337,B 24.9388,C -1.8069,E1 25.1405,E2 421.631} C_DIS
LIN {X 100.1637,Y 56.8287,Z 116,A 25.6365,B 24.9387,C -1.8089,E1 25.1386,E2 420.2306} C_DIS
LIN {X 98.7781,Y 59.2053,Z 116,A 26.9976,B 24.9384,C -1.8123,E1 25.1366,E2 418.8687} C_DIS
LIN {X 96.9931,Y 62.0826,Z 116,A 28.6006,B 24.9384,C -1.813,E1 25.1342,E2 417.2721} C_DIS
LIN {X 95.7118,Y 64.0433,Z 116,A 29.8315,B 24.938,C -1.819,E1 25.1323,E2 416.033} C_DIS
LIN {X 94.1112,Y 66.3729,Z 116,A 31.2302,B 24.9378,C -1.8222,E1 25.1301,E2 414.6336} C_DIS
LIN {X 92.454,Y 68.6625,Z 116,A 32.5951,B 24.9376,C -1.8238,E1 25.1278,E2 413.2715} C_DIS
LIN {X 90.7879,Y 70.8516,Z 116,A 34.0226,B 24.9372,C -1.8299,E1 25.1254,E2 411.8364} C_DIS
LIN {X 88.9735,Y 73.1163,Z 116,A 35.393,B 24.9372,C -1.8299,E1 25.123,E2 410.4722} C_DIS
LIN {X 86.9682,Y 75.4887,Z 116,A 36.8474,B 24.9372,C -1.8294,E1 25.1204,E2 409.0257} C_DIS
LIN {X 85.2787,Y 77.3939,Z 116,A 38.2252,B 24.9367,C -1.8374,E1 25.1178,E2 407.6352} C_DIS
LIN {X 83.406,Y 79.4092,Z 116,A 39.7486,B 24.936,C -1.8476,E1 25.1148,E2 406.0944} C_DIS
LIN {X 80.9848,Y 81.8739,Z 116,A 41.3323,B 24.9362,C -1.8451,E1 25.1117,E2 404.5233} C_DIS
LIN {X 78.3241,Y 84.4252,Z 116,A 43.1246,B 24.9361,C -1.847,E1 25.1081,E2 402.7339} C_DIS
LIN {X 76.2854,Y 86.2724,Z 116,A 44.6543,B 24.9353,C -1.8571,E1 25.1049,E2 401.1864} C_DIS
LIN {X 74.0872,Y 88.1667,Z 116,A 45.9253,B 24.9357,C -1.852,E1 25.1022,E2 399.9324} C_DIS
LIN {X 71.9603,Y 89.9116,Z 116,A 47.3207,B 24.9354,C -1.8558,E1 25.0992,E2 398.5333} C_DIS
LIN {X 69.7321,Y 91.6505,Z 116,A 48.8461,B 24.9349,C -1.8638,E1 25.0958,E2 396.9946} C_DIS
LIN {X 67.4005,Y 93.378,Z 116,A 50.1275,B 24.9352,C -1.859,E1 25.0929,E2 395.7291} C_DIS
LIN {X 65.0886,Y 95.004,Z 116,A 51.5287,B 24.9351,C -1.8611,E1 25.0897,E2 394.3277} C_DIS
LIN {X 62.8009,Y 96.532,Z 116,A 53.0482,B 24.9344,C -1.8702,E1 25.0861,E2 392.7918} C_DIS
LIN {X 60.1268,Y 98.2181,Z 116,A 54.31,B 24.9353,C -1.8585,E1 25.0832,E2 391.5615} C_DIS
LIN {X 57.9887,Y 99.4972,Z 116,A 55.696,B 24.9347,C -1.867,E1 25.0798,E2 390.1599} C_DIS
LIN {X 55.4631,Y 100.9263,Z 116,A 57.1014,B 24.9347,C -1.8673,E1 25.0764,E2 388.7579} C_DIS
LIN {X 52.9696,Y 102.257,Z 116,A 58.5378,B 24.9344,C -1.8705,E1 25.0728,E2 387.3178} C_DIS
LIN {X 50.4441,Y 103.5262,Z 116,A 59.9401,B 24.9344,C -1.8721,E1 25.0693,E2 385.9155} C_DIS
LIN {X 47.8883,Y 104.733,Z 116,A 61.3428,B 24.9342,C -1.8736,E1 25.0658,E2 384.5128} C_DIS
LIN {X 44.873,Y 106.0581,Z 116,A 62.7335,B 24.9348,C -1.8644,E1 25.0623,E2 383.1473} C_DIS
LIN {X 42.6916,Y 106.9566,Z 116,A 64.1489,B 24.934,C -1.8764,E1 25.0585,E2 381.7068} C_DIS
LIN {X 40.1247,Y 107.9462,Z 116,A 65.5467,B 24.9338,C -1.879,E1 25.0549,E2 380.3058} C_DIS
LIN {X 37.1913,Y 108.9902,Z 116,A 66.9314,B 24.9342,C -1.873,E1 25.0513,E2 378.9379} C_DIS
LIN {X 34.7797,Y 109.785,Z 116,A 68.3541,B 24.9337,C -1.8811,E1 25.0475,E2 377.4987} C_DIS
LIN {X 32.0024,Y 110.6261,Z 116,A 69.7296,B 24.9338,C -1.8792,E1 25.0438,E2 376.1303} C_DIS
LIN {X 29.1356,Y 111.4147,Z 116,A 71.1787,B 24.9338,C -1.8788,E1 25.0399,E2 374.6843} C_DIS
LIN {X 26.6092,Y 112.0461,Z 116,A 72.5672,B 24.9335,C -1.8836,E1 25.0361,E2 373.2863} C_DIS
LIN {X 23.8514,Y 112.6654,Z 116,A 74.045,B 24.9332,C -1.8875,E1 25.032,E2 371.8014} C_DIS
LIN {X 20.478,Y 113.325,Z 116,A 75.4276,B 24.9342,C -1.8738,E1 25.0284,E2 370.4527} C_DIS
LIN {X 17.8798,Y 113.7641,Z 116,A 76.8144,B 24.9339,C -1.8776,E1 25.0245,E2 369.0584} C_DIS
LIN {X 15.4986,Y 114.1147,Z 116,A 78.1554,B 24.9335,C -1.8842,E1 25.0208,E2 367.7031} C_DIS
Enddeposition()
END
